LIN {X 0,Y 314.247,Z 438.29,A -85,B 0,C 180,E1 -15747.116,E2 -15747.116} C_VEL
LIN {X 0,Y 313.392,Z 444.97,A -85,B 0,C 180,E1 -15749.358,E2 -15749.358} C_VEL
LIN {X 0,Y 312.88,Z 449.381,A -85,B 0,C 180,E1 -15751.288,E2 -15751.288} C_VEL
LIN {X 0,Y 312.504,Z 451.733,A -85,B 0,C 180,E1 -15752.578,E2 -15752.578} C_VEL
LIN {X 0,Y 312.347,Z 453.646,A -85,B 0,C 180,E1 -15753.871,E2 -15753.871} C_VEL
LIN {X 0,Y 312.37,Z 455.131,A -85,B 0,C 180,E1 -15755.164,E2 -15755.164} C_VEL
LIN {X 0,Y 312.273,Z 456.882,A -85,B 0,C 180,E1 -15757.761,E2 -15757.761} C_VEL
LIN {X 0,Y 312.327,Z 457.191,A -85,B 0,C 180,E1 -15759.063,E2 -15759.063} C_VEL
LIN {X 0,Y 312.449,Z 457.109,A -85,B 0,C 180,E1 -15760.367,E2 -15760.367} C_VEL
LIN {X 0,Y 312.916,Z 455.702,A -85,B 0,C 180,E1 -15762.979,E2 -15762.979} C_VEL
LIN {X 0,Y 313.359,Z 454.404,A -85,B 0,C 180,E1 -15764.283,E2 -15764.283} C_VEL
LIN {X 0,Y 314.081,Z 451.635,A -85,B 0,C 180,E1 -15766.242,E2 -15766.242} C_VEL
LIN {X 0,Y 314.982,Z 447.824,A -85,B 0,C 180,E1 -15768.202,E2 -15768.202} C_VEL
LIN {X 0,Y 316.106,Z 442.855,A -85,B 0,C 180,E1 -15770.158,E2 -15770.158} C_VEL
LIN {X 0,Y 317.523,Z 436.525,A -85,B 0,C 180,E1 -15772.103,E2 -15772.103} C_VEL
LIN {X 0,Y 319.103,Z 428.554,A -85,B 0,C 180,E1 -15774.045,E2 -15774.045} C_VEL
LIN {X 0,Y 320.652,Z 420.359,A -85,B 0,C 180,E1 -15775.65,E2 -15775.65} C_VEL
LIN {X 0,Y 322.026,Z 411.372,A -85,B 0,C 180,E1 -15777.102,E2 -15777.102} C_VEL
LIN {X 0,Y 323.472,Z 401.574,A -85,B 0,C 180,E1 -15778.377,E2 -15778.377} C_VEL
LIN {X 0,Y 324.734,Z 390.84,A -85,B 0,C 180,E1 -15779.496,E2 -15779.496} C_VEL
LIN {X 0,Y 325.769,Z 379.701,A -85,B 0,C 180,E1 -15780.403,E2 -15780.403} C_VEL
LIN {X 0,Y 326.491,Z 366.602,A -85,B 0,C 180,E1 -15781.205,E2 -15781.205} C_VEL
LIN {X 0,Y 326.866,Z 354.631,A -85,B 0,C 180,E1 -15781.696,E2 -15781.696} C_VEL
LIN {X 0,Y 327.637,Z 314.685,A -85,B 0,C 180,E1 -15782.625,E2 -15782.625} C_VEL
LIN {X 0,Y 328.12,Z 297.79,A -85,B 0,C 180,E1 -15782.993,E2 -15782.993} C_VEL
LIN {X 0,Y 320.551,Z 282.248,A -85,B 0,C 180,E1 -15784.14,E2 -15784.14} C_VEL
LIN {X 0,Y 313.584,Z 269.449,A -85,B 0,C 180,E1 -15785.22,E2 -15785.22} C_VEL
LIN {X 0,Y 312.651,Z 267.172,A -85,B 0,C 180,E1 -15785.452,E2 -15785.452} C_VEL
LIN {X 0,Y 312.55,Z 266.564,A -85,B 0,C 180,E1 -15785.777,E2 -15785.777} C_VEL
LIN {X 0,Y 312.477,Z 266.546,A -85,B 0,C 180,E1 -15789.032,E2 -15789.032} C_VEL
LIN {X 0,Y 312.456,Z 266.549,A -85,B 0,C 180,E1 -15792.188,E2 -15792.188} C_VEL
LIN {X 0,Y 311.815,Z 266.64,A -85,B 0,C 180,E1 -15793.264,E2 -15793.264} C_VEL
LIN {X 0,Y 308.975,Z 266.996,A -85,B 0,C 180,E1 -15795.016,E2 -15795.016} C_VEL
LIN {X 0,Y 306.549,Z 267.286,A -85,B 0,C 180,E1 -15796.436,E2 -15796.436} C_VEL
LIN {X 0,Y 305.5,Z 267.412,A -85,B 0,C 180,E1 -15797.536,E2 -15797.536} C_VEL
LIN {X 0,Y 305.412,Z 267.426,A -85,B 0,C 180,E1 -15797.908,E2 -15797.908} C_VEL
LIN {X 0,Y 305.44,Z 267.414,A -85,B 0,C 180,E1 -15801.592,E2 -15801.592} C_VEL
LIN {X 0,Y 305.46,Z 267.432,A -85,B 0,C 180,E1 -15804.886,E2 -15804.886} C_VEL
LIN {X 0,Y 305.44,Z 267.41,A -85,B 0,C 180,E1 -15808.358,E2 -15808.358} C_VEL
LIN {X 0,Y 305.463,Z 267.41,A -85,B 0,C 180,E1 -15811.107,E2 -15811.107} C_VEL
LIN {X 0,Y 305.497,Z 267.433,A -85,B 0,C 180,E1 -15814.081,E2 -15814.081} C_VEL
LIN {X 0,Y 305.471,Z 267.395,A -85,B 0,C 180,E1 -15816.975,E2 -15816.975} C_VEL
LIN {X 0,Y 305.576,Z 267.413,A -85,B 0,C 180,E1 -15821.216,E2 -15821.216} C_VEL
LIN {X 0,Y 305.646,Z 267.399,A -85,B 0,C 180,E1 -15825.348,E2 -15825.348} C_VEL
LIN {X 0,Y 305.62,Z 267.409,A -85,B 0,C 180,E1 -15829.399,E2 -15829.399} C_VEL
LIN {X 0,Y 305.741,Z 267.394,A -85,B 0,C 180,E1 -15832.072,E2 -15832.072} C_VEL
LIN {X 0,Y 305.65,Z 267.407,A -85,B 0,C 180,E1 -15834.722,E2 -15834.722} C_VEL
LIN {X 0,Y 305.941,Z 267.374,A -85,B 0,C 180,E1 -15838.683,E2 -15838.683} C_VEL
LIN {X 0,Y 305.93,Z 267.364,A -85,B 0,C 180,E1 -15841.316,E2 -15841.316} C_VEL
LIN {X 0,Y 305.654,Z 267.412,A -85,B 0,C 180,E1 -15845.277,E2 -15845.277} C_VEL
LIN {X 0,Y 305.74,Z 267.387,A -85,B 0,C 180,E1 -15847.927,E2 -15847.927} C_VEL
LIN {X 0,Y 305.592,Z 267.41,A -85,B 0,C 180,E1 -15851.945,E2 -15851.945} C_VEL
LIN {X 0,Y 305.604,Z 267.414,A -85,B 0,C 180,E1 -15855.014,E2 -15855.014} C_VEL
LIN {X 0,Y 305.542,Z 267.425,A -85,B 0,C 180,E1 -15859.428,E2 -15859.428} C_VEL
LIN {X 0,Y 305.483,Z 267.429,A -85,B 0,C 180,E1 -15863.039,E2 -15863.039} C_VEL
LIN {X 0,Y 305.463,Z 267.419,A -85,B 0,C 180,E1 -15866.196,E2 -15866.196} C_VEL
LIN {X 0,Y 305.419,Z 267.425,A -85,B 0,C 180,E1 -15869.025,E2 -15869.025} C_VEL
LIN {X 0,Y 305.431,Z 267.435,A -85,B 0,C 180,E1 -15871.953,E2 -15871.953} C_VEL
LIN {X 0,Y 305.458,Z 267.424,A -85,B 0,C 180,E1 -15875.114,E2 -15875.114} C_VEL
LIN {X 0,Y 305.43,Z 267.426,A -85,B 0,C 180,E1 -15878.525,E2 -15878.525} C_VEL
LIN {X 0,Y 305.431,Z 267.431,A -85,B 0,C 180,E1 -15882.581,E2 -15882.581} C_VEL
LIN {X 0,Y 305.418,Z 267.433,A -85,B 0,C 180,E1 -15886.344,E2 -15886.344} C_VEL
LIN {X 0,Y 305.466,Z 267.601,A -85,B 0,C 180,E1 -15890.617,E2 -15890.617} C_VEL
LIN {X 0,Y 308.864,Z 279.639,A -85,B 0,C 180,E1 -15894.049,E2 -15894.049} C_VEL
LIN {X 0,Y 311.517,Z 290.832,A -85,B 0,C 180,E1 -15896.979,E2 -15896.979} C_VEL
LIN {X 0,Y 313.244,Z 300.295,A -85,B 0,C 180,E1 -15899.308,E2 -15899.308} C_VEL
LIN {X 0,Y 311.503,Z 313.167,A -85,B 0,C 180,E1 -15902.016,E2 -15902.016} C_VEL
LIN {X 0,Y 311.73,Z 315.517,A -85,B 0,C 180,E1 -15902.182,E2 -15902.182} C_VEL
LIN {X 0,Y 316.099,Z 342.071,A -85,B 0,C 180,E1 -15903.321,E2 -15903.321} C_VEL
LIN {X 0,Y 319.329,Z 367.742,A -85,B 0,C 180,E1 -15904.287,E2 -15904.287} C_VEL
LIN {X 0,Y 319.905,Z 376.948,A -85,B 0,C 180,E1 -15904.572,E2 -15904.572} C_VEL
LIN {X 0,Y 318.499,Z 425.443,A -85,B 0,C 180,E1 -15905.69,E2 -15905.69} C_VEL
LIN {X 0,Y 317.484,Z 439.253,A -85,B 0,C 180,E1 -15906.259,E2 -15906.259} C_VEL
LIN {X 0,Y 316.086,Z 451.686,A -85,B 0,C 180,E1 -15907.015,E2 -15907.015} C_VEL
LIN {X 0,Y 314.257,Z 463.613,A -85,B 0,C 180,E1 -15908.001,E2 -15908.001} C_VEL
LIN {X 0,Y 312.257,Z 475.089,A -85,B 0,C 180,E1 -15909.238,E2 -15909.238} C_VEL
LIN {X 0,Y 310.326,Z 485.479,A -85,B 0,C 180,E1 -15910.657,E2 -15910.657} C_VEL
LIN {X 0,Y 308.647,Z 494.011,A -85,B 0,C 180,E1 -15912.097,E2 -15912.097} C_VEL
LIN {X 0,Y 306.953,Z 503.327,A -85,B 0,C 180,E1 -15914.053,E2 -15914.053} C_VEL
LIN {X 0,Y 305.899,Z 509.739,A -85,B 0,C 180,E1 -15915.701,E2 -15915.701} C_VEL
LIN {X 0,Y 304.737,Z 516.994,A -85,B 0,C 180,E1 -15918.02,E2 -15918.02} C_VEL
LIN {X 0,Y 304.214,Z 521.881,A -85,B 0,C 180,E1 -15920.022,E2 -15920.022} C_VEL
LIN {X 0,Y 304.081,Z 525.679,A -85,B 0,C 180,E1 -15922.029,E2 -15922.029} C_VEL
LIN {X 0,Y 304.187,Z 527.793,A -85,B 0,C 180,E1 -15923.454,E2 -15923.454} C_VEL
LIN {X 0,Y 304.482,Z 530.322,A -85,B 0,C 180,E1 -15926.029,E2 -15926.029} C_VEL
LIN {X 0,Y 304.663,Z 531.039,A -85,B 0,C 180,E1 -15927.355,E2 -15927.355} C_VEL
LIN {X 0,Y 304.672,Z 531.334,A -85,B 0,C 180,E1 -15928.678,E2 -15928.678} C_VEL
LIN {X 0,Y 304.795,Z 531.2,A -85,B 0,C 180,E1 -15929.999,E2 -15929.999} C_VEL
LIN {X 0,Y 304.732,Z 530.624,A -85,B 0,C 180,E1 -15931.321,E2 -15931.321} C_VEL
LIN {X 0,Y 304.731,Z 529.649,A -85,B 0,C 180,E1 -15932.643,E2 -15932.643} C_VEL
LIN {X 0,Y 304.622,Z 528.244,A -85,B 0,C 180,E1 -15933.968,E2 -15933.968} C_VEL
LIN {X 0,Y 304.391,Z 525.237,A -85,B 0,C 180,E1 -15935.963,E2 -15935.963} C_VEL
LIN {X 0,Y 304.244,Z 521.148,A -85,B 0,C 180,E1 -15937.966,E2 -15937.966} C_VEL
LIN {X 0,Y 304.376,Z 514.864,A -85,B 0,C 180,E1 -15940.308,E2 -15940.308} C_VEL
LIN {X 0,Y 304.867,Z 508.012,A -85,B 0,C 180,E1 -15942.311,E2 -15942.311} C_VEL
LIN {X 0,Y 305.704,Z 499.529,A -85,B 0,C 180,E1 -15944.307,E2 -15944.307} C_VEL
LIN {X 0,Y 306.686,Z 490.83,A -85,B 0,C 180,E1 -15945.961,E2 -15945.961} C_VEL
LIN {X 0,Y 307.809,Z 481.296,A -85,B 0,C 180,E1 -15947.437,E2 -15947.437} C_VEL
LIN {X 0,Y 309.296,Z 469.516,A -85,B 0,C 180,E1 -15948.892,E2 -15948.892} C_VEL
LIN {X 0,Y 310.641,Z 457.868,A -85,B 0,C 180,E1 -15950.009,E2 -15950.009} C_VEL
LIN {X 0,Y 311.816,Z 445.781,A -85,B 0,C 180,E1 -15950.878,E2 -15950.878} C_VEL
LIN {X 0,Y 312.673,Z 432.658,A -85,B 0,C 180,E1 -15951.552,E2 -15951.552} C_VEL
LIN {X 0,Y 313.184,Z 420.288,A -85,B 0,C 180,E1 -15951.947,E2 -15951.947} C_VEL
LIN {X 0,Y 313.933,Z 371.708,A -85,B 0,C 180,E1 -15953.054,E2 -15953.054} C_VEL
LIN {X 0,Y 309.351,Z 325.296,A -85,B 0,C 180,E1 -15954.472,E2 -15954.472} C_VEL
LIN {X 0,Y 308.185,Z 315.1,A -85,B 0,C 180,E1 -15954.851,E2 -15954.851} C_VEL
LIN {X 0,Y 310.188,Z 295.934,A -85,B 0,C 180,E1 -15958.78,E2 -15958.78} C_VEL
LIN {X 0,Y 310.465,Z 290.771,A -85,B 0,C 180,E1 -15959.867,E2 -15959.867} C_VEL
LIN {X 0,Y 307.511,Z 276.202,A -85,B 0,C 180,E1 -15963.263,E2 -15963.263} C_VEL
LIN {X 0,Y 305.499,Z 267.537,A -85,B 0,C 180,E1 -15965.435,E2 -15965.435} C_VEL
LIN {X 0,Y 305.428,Z 267.433,A -85,B 0,C 180,E1 -15968.524,E2 -15968.524} C_VEL
LIN {X 0,Y 305.428,Z 267.439,A -85,B 0,C 180,E1 -15972.58,E2 -15972.58} C_VEL
LIN {X 0,Y 305.413,Z 267.431,A -85,B 0,C 180,E1 -15976.343,E2 -15976.343} C_VEL
LIN {X 0,Y 305.402,Z 267.44,A -85,B 0,C 180,E1 -15979.884,E2 -15979.884} C_VEL
LIN {X 0,Y 305.454,Z 267.435,A -85,B 0,C 180,E1 -15983.636,E2 -15983.636} C_VEL
LIN {X 0,Y 305.455,Z 267.433,A -85,B 0,C 180,E1 -15986.482,E2 -15986.482} C_VEL
LIN {X 0,Y 305.407,Z 267.44,A -85,B 0,C 180,E1 -15989.585,E2 -15989.585} C_VEL
LIN {X 0,Y 305.444,Z 267.437,A -85,B 0,C 180,E1 -15992.601,E2 -15992.601} C_VEL
LIN {X 0,Y 305.463,Z 267.43,A -85,B 0,C 180,E1 -15995.535,E2 -15995.535} C_VEL
LIN {X 0,Y 305.451,Z 267.436,A -85,B 0,C 180,E1 -15998.399,E2 -15998.399} C_VEL
LIN {X 0,Y 305.525,Z 267.421,A -85,B 0,C 180,E1 -16002.6,E2 -16002.6} C_VEL
LIN {X 0,Y 305.616,Z 267.414,A -85,B 0,C 180,E1 -16005.348,E2 -16005.348} C_VEL
LIN {X 0,Y 305.613,Z 267.408,A -85,B 0,C 180,E1 -16009.399,E2 -16009.399} C_VEL
LIN {X 0,Y 305.734,Z 267.395,A -85,B 0,C 180,E1 -16012.073,E2 -16012.073} C_VEL
LIN {X 0,Y 305.647,Z 267.414,A -85,B 0,C 180,E1 -16014.723,E2 -16014.723} C_VEL
LIN {X 0,Y 305.924,Z 267.37,A -85,B 0,C 180,E1 -16018.684,E2 -16018.684} C_VEL
LIN {X 0,Y 305.933,Z 267.371,A -85,B 0,C 180,E1 -16021.317,E2 -16021.317} C_VEL
LIN {X 0,Y 305.773,Z 267.392,A -85,B 0,C 180,E1 -16026.599,E2 -16026.599} C_VEL
LIN {X 0,Y 305.674,Z 267.399,A -85,B 0,C 180,E1 -16029.262,E2 -16029.262} C_VEL
LIN {X 0,Y 305.575,Z 267.418,A -85,B 0,C 180,E1 -16033.297,E2 -16033.297} C_VEL
LIN {X 0,Y 305.541,Z 267.423,A -85,B 0,C 180,E1 -16036.023,E2 -16036.023} C_VEL
LIN {X 0,Y 305.475,Z 267.433,A -85,B 0,C 180,E1 -16040.188,E2 -16040.188} C_VEL
LIN {X 0,Y 305.447,Z 267.432,A -85,B 0,C 180,E1 -16044.467,E2 -16044.467} C_VEL
LIN {X 0,Y 305.432,Z 267.433,A -85,B 0,C 180,E1 -16047.401,E2 -16047.401} C_VEL
LIN {X 0,Y 305.409,Z 267.441,A -85,B 0,C 180,E1 -16050.415,E2 -16050.415} C_VEL
LIN {X 0,Y 305.458,Z 267.432,A -85,B 0,C 180,E1 -16054.079,E2 -16054.079} C_VEL
LIN {X 0,Y 305.445,Z 267.435,A -85,B 0,C 180,E1 -16056.744,E2 -16056.744} C_VEL
LIN {X 0,Y 305.403,Z 267.432,A -85,B 0,C 180,E1 -16060.591,E2 -16060.591} C_VEL
LIN {X 0,Y 305.415,Z 267.421,A -85,B 0,C 180,E1 -16063.658,E2 -16063.658} C_VEL
LIN {X 0,Y 305.43,Z 267.438,A -85,B 0,C 180,E1 -16067.42,E2 -16067.42} C_VEL
LIN {X 0,Y 305.438,Z 267.428,A -85,B 0,C 180,E1 -16071.594,E2 -16071.594} C_VEL
LIN {X 0,Y 305.459,Z 267.43,A -85,B 0,C 180,E1 -16074.888,E2 -16074.888} C_VEL
LIN {X 0,Y 305.437,Z 267.433,A -85,B 0,C 180,E1 -16078.361,E2 -16078.361} C_VEL
LIN {X 0,Y 305.449,Z 267.431,A -85,B 0,C 180,E1 -16081.108,E2 -16081.108} C_VEL
LIN {X 0,Y 305.478,Z 267.428,A -85,B 0,C 180,E1 -16084.081,E2 -16084.081} C_VEL
LIN {X 0,Y 305.456,Z 267.433,A -85,B 0,C 180,E1 -16088.401,E2 -16088.401} C_VEL
LIN {X 0,Y 305.5,Z 267.401,A -85,B 0,C 180,E1 -16091.213,E2 -16091.213} C_VEL
LIN {X 0,Y 305.528,Z 267.629,A -85,B 0,C 180,E1 -16093.45,E2 -16093.45} C_VEL
LIN {X 0,Y 305.832,Z 268.784,A -85,B 0,C 180,E1 -16093.661,E2 -16093.661} C_VEL
LIN {X 0,Y 314.272,Z 288.888,A -85,B 0,C 180,E1 -16094.778,E2 -16094.778} C_VEL
LIN {X 0,Y 315.387,Z 291.963,A -85,B 0,C 180,E1 -16094.93,E2 -16094.93} C_VEL
LIN {X 0,Y 314.323,Z 354.388,A -85,B 0,C 180,E1 -16096.373,E2 -16096.373} C_VEL
LIN {X 0,Y 313.978,Z 367.298,A -85,B 0,C 180,E1 -16096.917,E2 -16096.917} C_VEL
LIN {X 0,Y 313.505,Z 379.756,A -85,B 0,C 180,E1 -16097.705,E2 -16097.705} C_VEL
LIN {X 0,Y 312.674,Z 391.136,A -85,B 0,C 180,E1 -16098.658,E2 -16098.658} C_VEL
LIN {X 0,Y 311.574,Z 402.813,A -85,B 0,C 180,E1 -16099.933,E2 -16099.933} C_VEL
LIN {X 0,Y 310.555,Z 413.216,A -85,B 0,C 180,E1 -16101.378,E2 -16101.378} C_VEL
LIN {X 0,Y 309.377,Z 423.453,A -85,B 0,C 180,E1 -16103.151,E2 -16103.151} C_VEL
LIN {X 0,Y 308.236,Z 432.34,A -85,B 0,C 180,E1 -16105.096,E2 -16105.096} C_VEL
LIN {X 0,Y 307.228,Z 439.521,A -85,B 0,C 180,E1 -16107.05,E2 -16107.05} C_VEL
LIN {X 0,Y 306.348,Z 446.095,A -85,B 0,C 180,E1 -16109.343,E2 -16109.343} C_VEL
LIN {X 0,Y 305.811,Z 450.446,A -85,B 0,C 180,E1 -16111.317,E2 -16111.317} C_VEL
LIN {X 0,Y 305.442,Z 452.767,A -85,B 0,C 180,E1 -16112.638,E2 -16112.638} C_VEL
LIN {X 0,Y 305.298,Z 454.65,A -85,B 0,C 180,E1 -16113.96,E2 -16113.96} C_VEL
LIN {X 0,Y 305.317,Z 456.082,A -85,B 0,C 180,E1 -16115.283,E2 -16115.283} C_VEL
LIN {X 0,Y 305.243,Z 457.776,A -85,B 0,C 180,E1 -16117.941,E2 -16117.941} C_VEL
LIN {X 0,Y 305.304,Z 458.059,A -85,B 0,C 180,E1 -16119.273,E2 -16119.273} C_VEL
LIN {X 0,Y 305.457,Z 457.922,A -85,B 0,C 180,E1 -16120.607,E2 -16120.607} C_VEL
LIN {X 0,Y 305.96,Z 456.46,A -85,B 0,C 180,E1 -16123.28,E2 -16123.28} C_VEL
LIN {X 0,Y 306.433,Z 455.132,A -85,B 0,C 180,E1 -16124.613,E2 -16124.613} C_VEL
LIN {X 0,Y 307.192,Z 452.307,A -85,B 0,C 180,E1 -16126.617,E2 -16126.617} C_VEL
LIN {X 0,Y 308.169,Z 448.433,A -85,B 0,C 180,E1 -16128.619,E2 -16128.619} C_VEL
LIN {X 0,Y 309.397,Z 443.38,A -85,B 0,C 180,E1 -16130.615,E2 -16130.615} C_VEL
LIN {X 0,Y 310.889,Z 436.95,A -85,B 0,C 180,E1 -16132.601,E2 -16132.601} C_VEL
LIN {X 0,Y 312.574,Z 428.89,A -85,B 0,C 180,E1 -16134.58,E2 -16134.58} C_VEL
LIN {X 0,Y 314.186,Z 420.657,A -85,B 0,C 180,E1 -16136.205,E2 -16136.205} C_VEL
LIN {X 0,Y 315.683,Z 411.474,A -85,B 0,C 180,E1 -16137.693,E2 -16137.693} C_VEL
LIN {X 0,Y 317.115,Z 401.452,A -85,B 0,C 180,E1 -16138.999,E2 -16138.999} C_VEL
LIN {X 0,Y 318.507,Z 390.466,A -85,B 0,C 180,E1 -16140.132,E2 -16140.132} C_VEL
LIN {X 0,Y 319.526,Z 379.515,A -85,B 0,C 180,E1 -16141.019,E2 -16141.019} C_VEL
LIN {X 0,Y 320.249,Z 366.514,A -85,B 0,C 180,E1 -16141.811,E2 -16141.811} C_VEL
LIN {X 0,Y 320.628,Z 354.436,A -85,B 0,C 180,E1 -16142.291,E2 -16142.291} C_VEL
LIN {X 0,Y 321.455,Z 314.337,A -85,B 0,C 180,E1 -16143.234,E2 -16143.234} C_VEL
LIN {X 0,Y 321.851,Z 299.831,A -85,B 0,C 180,E1 -16143.56,E2 -16143.56} C_VEL
LIN {X 0,Y 313.661,Z 283.186,A -85,B 0,C 180,E1 -16144.849,E2 -16144.849} C_VEL
LIN {X 0,Y 306.731,Z 270.599,A -85,B 0,C 180,E1 -16145.968,E2 -16145.968} C_VEL
LIN {X 0,Y 305.602,Z 268.05,A -85,B 0,C 180,E1 -16146.239,E2 -16146.239} C_VEL
LIN {X 0,Y 305.49,Z 267.483,A -85,B 0,C 180,E1 -16146.493,E2 -16146.493} C_VEL
LIN {X 0,Y 305.41,Z 267.446,A -85,B 0,C 180,E1 -16150.115,E2 -16150.115} C_VEL
LIN {X 0,Y 305.42,Z 267.44,A -85,B 0,C 180,E1 -16153.656,E2 -16153.656} C_VEL
LIN {X 0,Y 305.433,Z 267.419,A -85,B 0,C 180,E1 -16157.418,E2 -16157.418} C_VEL
LIN {X 0,Y 305.412,Z 267.426,A -85,B 0,C 180,E1 -16157.908,E2 -16157.908} C_VEL
LIN {X 0,Y 304.742,Z 267.525,A -85,B 0,C 180,E1 -16159.009,E2 -16159.009} C_VEL
LIN {X 0,Y 301.912,Z 267.865,A -85,B 0,C 180,E1 -16160.801,E2 -16160.801} C_VEL
LIN {X 0,Y 299.516,Z 268.151,A -85,B 0,C 180,E1 -16162.255,E2 -16162.255} C_VEL
LIN {X 0,Y 298.488,Z 268.279,A -85,B 0,C 180,E1 -16163.38,E2 -16163.38} C_VEL
LIN {X 0,Y 298.403,Z 268.294,A -85,B 0,C 180,E1 -16163.761,E2 -16163.761} C_VEL
LIN {X 0,Y 298.391,Z 268.308,A -85,B 0,C 180,E1 -16167.199,E2 -16167.199} C_VEL
LIN {X 0,Y 298.369,Z 268.286,A -85,B 0,C 180,E1 -16170.635,E2 -16170.635} C_VEL
LIN {X 0,Y 298.436,Z 268.307,A -85,B 0,C 180,E1 -16174.919,E2 -16174.919} C_VEL
LIN {X 0,Y 298.401,Z 268.266,A -85,B 0,C 180,E1 -16177.862,E2 -16177.862} C_VEL
LIN {X 0,Y 298.522,Z 268.281,A -85,B 0,C 180,E1 -16180.755,E2 -16180.755} C_VEL
LIN {X 0,Y 298.59,Z 268.279,A -85,B 0,C 180,E1 -16184.994,E2 -16184.994} C_VEL
LIN {X 0,Y 298.579,Z 268.29,A -85,B 0,C 180,E1 -16189.146,E2 -16189.146} C_VEL
LIN {X 0,Y 298.693,Z 268.269,A -85,B 0,C 180,E1 -16191.884,E2 -16191.884} C_VEL
LIN {X 0,Y 298.62,Z 268.283,A -85,B 0,C 180,E1 -16194.598,E2 -16194.598} C_VEL
LIN {X 0,Y 298.907,Z 268.251,A -85,B 0,C 180,E1 -16198.652,E2 -16198.652} C_VEL
LIN {X 0,Y 298.898,Z 268.239,A -85,B 0,C 180,E1 -16201.347,E2 -16201.347} C_VEL
LIN {X 0,Y 298.727,Z 268.263,A -85,B 0,C 180,E1 -16206.755,E2 -16206.755} C_VEL
LIN {X 0,Y 298.621,Z 268.284,A -85,B 0,C 180,E1 -16209.482,E2 -16209.482} C_VEL
LIN {X 0,Y 298.539,Z 268.285,A -85,B 0,C 180,E1 -16213.616,E2 -16213.616} C_VEL
LIN {X 0,Y 298.483,Z 268.303,A -85,B 0,C 180,E1 -16216.412,E2 -16216.412} C_VEL
LIN {X 0,Y 298.482,Z 268.307,A -85,B 0,C 180,E1 -16219.641,E2 -16219.641} C_VEL
LIN {X 0,Y 298.416,Z 268.316,A -85,B 0,C 180,E1 -16223.601,E2 -16223.601} C_VEL
LIN {X 0,Y 298.402,Z 268.292,A -85,B 0,C 180,E1 -16226.583,E2 -16226.583} C_VEL
LIN {X 0,Y 298.352,Z 268.314,A -85,B 0,C 180,E1 -16229.648,E2 -16229.648} C_VEL
LIN {X 0,Y 298.388,Z 268.3,A -85,B 0,C 180,E1 -16232.801,E2 -16232.801} C_VEL
LIN {X 0,Y 298.401,Z 268.315,A -85,B 0,C 180,E1 -16236.072,E2 -16236.072} C_VEL
LIN {X 0,Y 298.371,Z 268.306,A -85,B 0,C 180,E1 -16239.492,E2 -16239.492} C_VEL
LIN {X 0,Y 298.366,Z 268.308,A -85,B 0,C 180,E1 -16243.097,E2 -16243.097} C_VEL
LIN {X 0,Y 298.367,Z 268.311,A -85,B 0,C 180,E1 -16246.915,E2 -16246.915} C_VEL
LIN {X 0,Y 298.413,Z 268.534,A -85,B 0,C 180,E1 -16249.912,E2 -16249.912} C_VEL
LIN {X 0,Y 301.837,Z 280.529,A -85,B 0,C 180,E1 -16253.445,E2 -16253.445} C_VEL
LIN {X 0,Y 304.446,Z 291.278,A -85,B 0,C 180,E1 -16256.356,E2 -16256.356} C_VEL
LIN {X 0,Y 306.43,Z 301.402,A -85,B 0,C 180,E1 -16258.933,E2 -16258.933} C_VEL
LIN {X 0,Y 305.149,Z 311.226,A -85,B 0,C 180,E1 -16261.075,E2 -16261.075} C_VEL
LIN {X 0,Y 305.001,Z 313.048,A -85,B 0,C 180,E1 -16261.364,E2 -16261.364} C_VEL
LIN {X 0,Y 309.751,Z 342.135,A -85,B 0,C 180,E1 -16262.671,E2 -16262.671} C_VEL
LIN {X 0,Y 312.825,Z 366.354,A -85,B 0,C 180,E1 -16263.617,E2 -16263.617} C_VEL
LIN {X 0,Y 313.654,Z 376.711,A -85,B 0,C 180,E1 -16263.965,E2 -16263.965} C_VEL
LIN {X 0,Y 312.216,Z 424.344,A -85,B 0,C 180,E1 -16265.08,E2 -16265.08} C_VEL
LIN {X 0,Y 311.17,Z 438.229,A -85,B 0,C 180,E1 -16265.658,E2 -16265.658} C_VEL
LIN {X 0,Y 309.71,Z 450.709,A -85,B 0,C 180,E1 -16266.425,E2 -16266.425} C_VEL
LIN {X 0,Y 307.92,Z 461.867,A -85,B 0,C 180,E1 -16267.346,E2 -16267.346} C_VEL
LIN {X 0,Y 305.849,Z 473.5,A -85,B 0,C 180,E1 -16268.605,E2 -16268.605} C_VEL
LIN {X 0,Y 303.846,Z 484.01,A -85,B 0,C 180,E1 -16270.052,E2 -16270.052} C_VEL
LIN {X 0,Y 301.881,Z 493.523,A -85,B 0,C 180,E1 -16271.682,E2 -16271.682} C_VEL
LIN {X 0,Y 300.097,Z 502.756,A -85,B 0,C 180,E1 -16273.678,E2 -16273.678} C_VEL
LIN {X 0,Y 298.736,Z 510.255,A -85,B 0,C 180,E1 -16275.698,E2 -16275.698} C_VEL
LIN {X 0,Y 297.757,Z 516.325,A -85,B 0,C 180,E1 -16277.735,E2 -16277.735} C_VEL
LIN {X 0,Y 297.159,Z 521.169,A -85,B 0,C 180,E1 -16279.783,E2 -16279.783} C_VEL
LIN {X 0,Y 297.013,Z 524.932,A -85,B 0,C 180,E1 -16281.838,E2 -16281.838} C_VEL
LIN {X 0,Y 297.124,Z 527.171,A -85,B 0,C 180,E1 -16283.435,E2 -16283.435} C_VEL
LIN {X 0,Y 297.397,Z 529.508,A -85,B 0,C 180,E1 -16285.934,E2 -16285.934} C_VEL
LIN {X 0,Y 297.613,Z 530.213,A -85,B 0,C 180,E1 -16287.292,E2 -16287.292} C_VEL
LIN {X 0,Y 297.622,Z 530.486,A -85,B 0,C 180,E1 -16288.646,E2 -16288.646} C_VEL
LIN {X 0,Y 297.747,Z 530.325,A -85,B 0,C 180,E1 -16289.999,E2 -16289.999} C_VEL
LIN {X 0,Y 297.682,Z 529.732,A -85,B 0,C 180,E1 -16291.352,E2 -16291.352} C_VEL
LIN {X 0,Y 297.682,Z 528.739,A -85,B 0,C 180,E1 -16292.706,E2 -16292.706} C_VEL
LIN {X 0,Y 297.553,Z 527.306,A -85,B 0,C 180,E1 -16294.063,E2 -16294.063} C_VEL
LIN {X 0,Y 297.281,Z 523.757,A -85,B 0,C 180,E1 -16296.382,E2 -16296.382} C_VEL
LIN {X 0,Y 297.162,Z 518.474,A -85,B 0,C 180,E1 -16298.842,E2 -16298.842} C_VEL
LIN {X 0,Y 297.4,Z 512.745,A -85,B 0,C 180,E1 -16300.897,E2 -16300.897} C_VEL
LIN {X 0,Y 297.951,Z 505.605,A -85,B 0,C 180,E1 -16302.948,E2 -16302.948} C_VEL
LIN {X 0,Y 298.705,Z 498.328,A -85,B 0,C 180,E1 -16304.65,E2 -16304.65} C_VEL
LIN {X 0,Y 299.834,Z 489.552,A -85,B 0,C 180,E1 -16306.335,E2 -16306.335} C_VEL
LIN {X 0,Y 301.053,Z 479.94,A -85,B 0,C 180,E1 -16307.841,E2 -16307.841} C_VEL
LIN {X 0,Y 302.362,Z 469.485,A -85,B 0,C 180,E1 -16309.166,E2 -16309.166} C_VEL
LIN {X 0,Y 303.728,Z 458.06,A -85,B 0,C 180,E1 -16310.308,E2 -16310.308} C_VEL
LIN {X 0,Y 304.948,Z 446.418,A -85,B 0,C 180,E1 -16311.194,E2 -16311.194} C_VEL
LIN {X 0,Y 305.869,Z 432.974,A -85,B 0,C 180,E1 -16311.923,E2 -16311.923} C_VEL
LIN {X 0,Y 306.457,Z 419.843,A -85,B 0,C 180,E1 -16312.366,E2 -16312.366} C_VEL
LIN {X 0,Y 307.263,Z 372.556,A -85,B 0,C 180,E1 -16313.465,E2 -16313.465} C_VEL
LIN {X 0,Y 302.775,Z 326.508,A -85,B 0,C 180,E1 -16314.91,E2 -16314.91} C_VEL
LIN {X 0,Y 301.342,Z 314.336,A -85,B 0,C 180,E1 -16315.35,E2 -16315.35} C_VEL
LIN {X 0,Y 303.309,Z 296.361,A -85,B 0,C 180,E1 -16319.115,E2 -16319.115} C_VEL
LIN {X 0,Y 303.6,Z 292.938,A -85,B 0,C 180,E1 -16319.847,E2 -16319.847} C_VEL
LIN {X 0,Y 301.035,Z 279.672,A -85,B 0,C 180,E1 -16322.991,E2 -16322.991} C_VEL
LIN {X 0,Y 298.495,Z 268.452,A -85,B 0,C 180,E1 -16325.832,E2 -16325.832} C_VEL
LIN {X 0,Y 298.368,Z 268.308,A -85,B 0,C 180,E1 -16329.491,E2 -16329.491} C_VEL
LIN {X 0,Y 298.363,Z 268.316,A -85,B 0,C 180,E1 -16333.096,E2 -16333.096} C_VEL
LIN {X 0,Y 298.362,Z 268.312,A -85,B 0,C 180,E1 -16336.914,E2 -16336.914} C_VEL
LIN {X 0,Y 298.377,Z 268.315,A -85,B 0,C 180,E1 -16341.01,E2 -16341.01} C_VEL
LIN {X 0,Y 298.396,Z 268.314,A -85,B 0,C 180,E1 -16343.927,E2 -16343.927} C_VEL
LIN {X 0,Y 298.383,Z 268.309,A -85,B 0,C 180,E1 -16347.198,E2 -16347.198} C_VEL
LIN {X 0,Y 298.396,Z 268.313,A -85,B 0,C 180,E1 -16351.898,E2 -16351.898} C_VEL
LIN {X 0,Y 298.428,Z 268.306,A -85,B 0,C 180,E1 -16354.919,E2 -16354.919} C_VEL
LIN {X 0,Y 298.389,Z 268.314,A -85,B 0,C 180,E1 -16357.861,E2 -16357.861} C_VEL
LIN {X 0,Y 298.453,Z 268.304,A -85,B 0,C 180,E1 -16360.751,E2 -16360.751} C_VEL
LIN {X 0,Y 298.577,Z 268.294,A -85,B 0,C 180,E1 -16364.994,E2 -16364.994} C_VEL
LIN {X 0,Y 298.572,Z 268.285,A -85,B 0,C 180,E1 -16369.146,E2 -16369.146} C_VEL
LIN {X 0,Y 298.686,Z 268.272,A -85,B 0,C 180,E1 -16371.884,E2 -16371.884} C_VEL
LIN {X 0,Y 298.616,Z 268.29,A -85,B 0,C 180,E1 -16374.598,E2 -16374.598} C_VEL
LIN {X 0,Y 298.892,Z 268.245,A -85,B 0,C 180,E1 -16378.653,E2 -16378.653} C_VEL
LIN {X 0,Y 298.9,Z 268.247,A -85,B 0,C 180,E1 -16381.348,E2 -16381.348} C_VEL
LIN {X 0,Y 298.721,Z 268.269,A -85,B 0,C 180,E1 -16386.756,E2 -16386.756} C_VEL
LIN {X 0,Y 298.607,Z 268.279,A -85,B 0,C 180,E1 -16389.483,E2 -16389.483} C_VEL
LIN {X 0,Y 298.534,Z 268.296,A -85,B 0,C 180,E1 -16393.617,E2 -16393.617} C_VEL
LIN {X 0,Y 298.474,Z 268.297,A -85,B 0,C 180,E1 -16396.413,E2 -16396.413} C_VEL
LIN {X 0,Y 298.433,Z 268.305,A -85,B 0,C 180,E1 -16399.617,E2 -16399.617} C_VEL
LIN {X 0,Y 298.38,Z 268.315,A -85,B 0,C 180,E1 -16403.605,E2 -16403.605} C_VEL
LIN {X 0,Y 298.393,Z 268.31,A -85,B 0,C 180,E1 -16406.584,E2 -16406.584} C_VEL
LIN {X 0,Y 298.349,Z 268.321,A -85,B 0,C 180,E1 -16409.649,E2 -16409.649} C_VEL
LIN {X 0,Y 298.386,Z 268.309,A -85,B 0,C 180,E1 -16412.802,E2 -16412.802} C_VEL
LIN {X 0,Y 298.397,Z 268.317,A -85,B 0,C 180,E1 -16416.073,E2 -16416.073} C_VEL
LIN {X 0,Y 298.368,Z 268.317,A -85,B 0,C 180,E1 -16419.493,E2 -16419.493} C_VEL
LIN {X 0,Y 298.364,Z 268.295,A -85,B 0,C 180,E1 -16423.098,E2 -16423.098} C_VEL
LIN {X 0,Y 298.365,Z 268.315,A -85,B 0,C 180,E1 -16426.916,E2 -16426.916} C_VEL
LIN {X 0,Y 298.382,Z 268.311,A -85,B 0,C 180,E1 -16431.012,E2 -16431.012} C_VEL
LIN {X 0,Y 298.401,Z 268.304,A -85,B 0,C 180,E1 -16433.929,E2 -16433.929} C_VEL
LIN {X 0,Y 298.39,Z 268.317,A -85,B 0,C 180,E1 -16437.201,E2 -16437.201} C_VEL
LIN {X 0,Y 298.361,Z 268.311,A -85,B 0,C 180,E1 -16440.64,E2 -16440.64} C_VEL
LIN {X 0,Y 298.421,Z 268.305,A -85,B 0,C 180,E1 -16444.919,E2 -16444.919} C_VEL
LIN {X 0,Y 298.39,Z 268.314,A -85,B 0,C 180,E1 -16447.862,E2 -16447.862} C_VEL
LIN {X 0,Y 298.451,Z 268.276,A -85,B 0,C 180,E1 -16450.752,E2 -16450.752} C_VEL
LIN {X 0,Y 298.488,Z 268.573,A -85,B 0,C 180,E1 -16452.947,E2 -16452.947} C_VEL
LIN {X 0,Y 298.719,Z 269.516,A -85,B 0,C 180,E1 -16453.123,E2 -16453.123} C_VEL
LIN {X 0,Y 306.932,Z 288.664,A -85,B 0,C 180,E1 -16454.244,E2 -16454.244} C_VEL
LIN {X 0,Y 308.831,Z 294.105,A -85,B 0,C 180,E1 -16454.516,E2 -16454.516} C_VEL
LIN {X 0,Y 307.644,Z 354.477,A -85,B 0,C 180,E1 -16455.932,E2 -16455.932} C_VEL
LIN {X 0,Y 307.311,Z 367.077,A -85,B 0,C 180,E1 -16456.452,E2 -16456.452} C_VEL
LIN {X 0,Y 306.837,Z 379.906,A -85,B 0,C 180,E1 -16457.265,E2 -16457.265} C_VEL
LIN {X 0,Y 305.958,Z 391.442,A -85,B 0,C 180,E1 -16458.238,E2 -16458.238} C_VEL
LIN {X 0,Y 304.963,Z 401.962,A -85,B 0,C 180,E1 -16459.377,E2 -16459.377} C_VEL
LIN {X 0,Y 303.832,Z 412.695,A -85,B 0,C 180,E1 -16460.85,E2 -16460.85} C_VEL
LIN {X 0,Y 302.862,Z 421.434,A -85,B 0,C 180,E1 -16462.333,E2 -16462.333} C_VEL
LIN {X 0,Y 301.603,Z 430.949,A -85,B 0,C 180,E1 -16464.317,E2 -16464.317} C_VEL
LIN {X 0,Y 300.468,Z 438.559,A -85,B 0,C 180,E1 -16466.313,E2 -16466.313} C_VEL
LIN {X 0,Y 299.519,Z 445.543,A -85,B 0,C 180,E1 -16468.656,E2 -16468.656} C_VEL
LIN {X 0,Y 298.943,Z 450.201,A -85,B 0,C 180,E1 -16470.674,E2 -16470.674} C_VEL
LIN {X 0,Y 298.381,Z 453.801,A -85,B 0,C 180,E1 -16472.701,E2 -16472.701} C_VEL
LIN {X 0,Y 298.248,Z 455.648,A -85,B 0,C 180,E1 -16474.054,E2 -16474.054} C_VEL
LIN {X 0,Y 298.252,Z 457.031,A -85,B 0,C 180,E1 -16475.409,E2 -16475.409} C_VEL
LIN {X 0,Y 298.199,Z 458.683,A -85,B 0,C 180,E1 -16478.161,E2 -16478.161} C_VEL
LIN {X 0,Y 298.287,Z 458.918,A -85,B 0,C 180,E1 -16479.493,E2 -16479.493} C_VEL
LIN {X 0,Y 298.68,Z 458.17,A -85,B 0,C 180,E1 -16482.227,E2 -16482.227} C_VEL
LIN {X 0,Y 299.012,Z 457.219,A -85,B 0,C 180,E1 -16483.594,E2 -16483.594} C_VEL
LIN {X 0,Y 299.976,Z 454.294,A -85,B 0,C 180,E1 -16486.141,E2 -16486.141} C_VEL
LIN {X 0,Y 301.017,Z 450.442,A -85,B 0,C 180,E1 -16488.373,E2 -16488.373} C_VEL
LIN {X 0,Y 302.207,Z 445.729,A -85,B 0,C 180,E1 -16490.416,E2 -16490.416} C_VEL
LIN {X 0,Y 303.685,Z 439.84,A -85,B 0,C 180,E1 -16492.408,E2 -16492.408} C_VEL
LIN {X 0,Y 305.412,Z 432.185,A -85,B 0,C 180,E1 -16494.469,E2 -16494.469} C_VEL
LIN {X 0,Y 307.348,Z 423.022,A -85,B 0,C 180,E1 -16496.397,E2 -16496.397} C_VEL
LIN {X 0,Y 308.919,Z 413.748,A -85,B 0,C 180,E1 -16497.983,E2 -16497.983} C_VEL
LIN {X 0,Y 310.501,Z 404.099,A -85,B 0,C 180,E1 -16499.306,E2 -16499.306} C_VEL
LIN {X 0,Y 311.871,Z 393.64,A -85,B 0,C 180,E1 -16500.467,E2 -16500.467} C_VEL
LIN {X 0,Y 313.032,Z 382.36,A -85,B 0,C 180,E1 -16501.443,E2 -16501.443} C_VEL
LIN {X 0,Y 313.838,Z 369.557,A -85,B 0,C 180,E1 -16502.276,E2 -16502.276} C_VEL
LIN {X 0,Y 314.327,Z 356.519,A -85,B 0,C 180,E1 -16502.848,E2 -16502.848} C_VEL
LIN {X 0,Y 315.288,Z 314.203,A -85,B 0,C 180,E1 -16503.867,E2 -16503.867} C_VEL
LIN {X 0,Y 315.607,Z 301.776,A -85,B 0,C 180,E1 -16504.155,E2 -16504.155} C_VEL
LIN {X 0,Y 306.347,Z 283.316,A -85,B 0,C 180,E1 -16505.667,E2 -16505.667} C_VEL
LIN {X 0,Y 299.695,Z 271.506,A -85,B 0,C 180,E1 -16506.786,E2 -16506.786} C_VEL
LIN {X 0,Y 298.519,Z 268.901,A -85,B 0,C 180,E1 -16507.082,E2 -16507.082} C_VEL
LIN {X 0,Y 298.416,Z 268.346,A -85,B 0,C 180,E1 -16507.354,E2 -16507.354} C_VEL
LIN {X 0,Y 298.347,Z 268.309,A -85,B 0,C 180,E1 -16511.268,E2 -16511.268} C_VEL
LIN {X 0,Y 298.355,Z 268.317,A -85,B 0,C 180,E1 -16515.034,E2 -16515.034} C_VEL
LIN {X 0,Y 298.347,Z 268.32,A -85,B 0,C 180,E1 -16518.921,E2 -16518.921} C_VEL
LIN {X 0,Y 298.385,Z 268.288,A -85,B 0,C 180,E1 -16522.237,E2 -16522.237} C_VEL
LIN {X 0,Y 298.403,Z 268.294,A -85,B 0,C 180,E1 -16523.761,E2 -16523.761} C_VEL
LIN {X 0,Y 297.722,Z 268.396,A -85,B 0,C 180,E1 -16524.888,E2 -16524.888} C_VEL
LIN {X 0,Y 294.83,Z 268.758,A -85,B 0,C 180,E1 -16526.723,E2 -16526.723} C_VEL
LIN {X 0,Y 292.397,Z 269.038,A -85,B 0,C 180,E1 -16528.212,E2 -16528.212} C_VEL
LIN {X 0,Y 291.377,Z 269.151,A -85,B 0,C 180,E1 -16529.366,E2 -16529.366} C_VEL
LIN {X 0,Y 291.307,Z 269.159,A -85,B 0,C 180,E1 -16529.757,E2 -16529.757} C_VEL
LIN {X 0,Y 291.348,Z 269.195,A -85,B 0,C 180,E1 -16533.191,E2 -16533.191} C_VEL
LIN {X 0,Y 291.363,Z 269.145,A -85,B 0,C 180,E1 -16537.298,E2 -16537.298} C_VEL
LIN {X 0,Y 291.456,Z 269.152,A -85,B 0,C 180,E1 -16540.27,E2 -16540.27} C_VEL
LIN {X 0,Y 291.538,Z 269.16,A -85,B 0,C 180,E1 -16544.634,E2 -16544.634} C_VEL
LIN {X 0,Y 291.525,Z 269.169,A -85,B 0,C 180,E1 -16548.88,E2 -16548.88} C_VEL
LIN {X 0,Y 291.646,Z 269.144,A -85,B 0,C 180,E1 -16551.686,E2 -16551.686} C_VEL
LIN {X 0,Y 291.59,Z 269.159,A -85,B 0,C 180,E1 -16554.467,E2 -16554.467} C_VEL
LIN {X 0,Y 291.874,Z 269.127,A -85,B 0,C 180,E1 -16558.62,E2 -16558.62} C_VEL
LIN {X 0,Y 291.866,Z 269.115,A -85,B 0,C 180,E1 -16561.379,E2 -16561.379} C_VEL
LIN {X 0,Y 291.679,Z 269.139,A -85,B 0,C 180,E1 -16566.919,E2 -16566.919} C_VEL
LIN {X 0,Y 291.564,Z 269.166,A -85,B 0,C 180,E1 -16569.714,E2 -16569.714} C_VEL
LIN {X 0,Y 291.51,Z 269.162,A -85,B 0,C 180,E1 -16573.951,E2 -16573.951} C_VEL
LIN {X 0,Y 291.437,Z 269.181,A -85,B 0,C 180,E1 -16576.821,E2 -16576.821} C_VEL
LIN {X 0,Y 291.421,Z 269.185,A -85,B 0,C 180,E1 -16579.86,E2 -16579.86} C_VEL
LIN {X 0,Y 291.355,Z 269.193,A -85,B 0,C 180,E1 -16584.209,E2 -16584.209} C_VEL
LIN {X 0,Y 291.327,Z 269.168,A -85,B 0,C 180,E1 -16587.281,E2 -16587.281} C_VEL
LIN {X 0,Y 291.297,Z 269.199,A -85,B 0,C 180,E1 -16590.441,E2 -16590.441} C_VEL
LIN {X 0,Y 291.34,Z 269.172,A -85,B 0,C 180,E1 -16593.699,E2 -16593.699} C_VEL
LIN {X 0,Y 291.35,Z 269.19,A -85,B 0,C 180,E1 -16597.248,E2 -16597.248} C_VEL
LIN {X 0,Y 291.297,Z 269.201,A -85,B 0,C 180,E1 -16600.648,E2 -16600.648} C_VEL
LIN {X 0,Y 291.279,Z 269.199,A -85,B 0,C 180,E1 -16604.404,E2 -16604.404} C_VEL
LIN {X 0,Y 291.292,Z 269.198,A -85,B 0,C 180,E1 -16608.412,E2 -16608.412} C_VEL
LIN {X 0,Y 291.348,Z 269.452,A -85,B 0,C 180,E1 -16609.152,E2 -16609.152} C_VEL
LIN {X 0,Y 294.082,Z 278.883,A -85,B 0,C 180,E1 -16612.058,E2 -16612.058} C_VEL
LIN {X 0,Y 296.77,Z 289.18,A -85,B 0,C 180,E1 -16615.001,E2 -16615.001} C_VEL
LIN {X 0,Y 299.275,Z 300.815,A -85,B 0,C 180,E1 -16618.102,E2 -16618.102} C_VEL
LIN {X 0,Y 299.585,Z 304.164,A -85,B 0,C 180,E1 -16618.929,E2 -16618.929} C_VEL
LIN {X 0,Y 298.573,Z 311.467,A -85,B 0,C 180,E1 -16620.527,E2 -16620.527} C_VEL
LIN {X 0,Y 299.421,Z 317.232,A -85,B 0,C 180,E1 -16620.852,E2 -16620.852} C_VEL
LIN {X 0,Y 303.948,Z 345.691,A -85,B 0,C 180,E1 -16622.143,E2 -16622.143} C_VEL
LIN {X 0,Y 307.001,Z 370.794,A -85,B 0,C 180,E1 -16623.137,E2 -16623.137} C_VEL
LIN {X 0,Y 307.383,Z 378.108,A -85,B 0,C 180,E1 -16623.369,E2 -16623.369} C_VEL
LIN {X 0,Y 305.934,Z 423.25,A -85,B 0,C 180,E1 -16624.441,E2 -16624.441} C_VEL
LIN {X 0,Y 304.996,Z 436.442,A -85,B 0,C 180,E1 -16624.995,E2 -16624.995} C_VEL
LIN {X 0,Y 303.411,Z 449.729,A -85,B 0,C 180,E1 -16625.814,E2 -16625.814} C_VEL
LIN {X 0,Y 301.397,Z 461.711,A -85,B 0,C 180,E1 -16626.828,E2 -16626.828} C_VEL
LIN {X 0,Y 299.222,Z 473.212,A -85,B 0,C 180,E1 -16628.107,E2 -16628.107} C_VEL
LIN {X 0,Y 297.175,Z 483.625,A -85,B 0,C 180,E1 -16629.584,E2 -16629.584} C_VEL
LIN {X 0,Y 295.118,Z 493.026,A -85,B 0,C 180,E1 -16631.247,E2 -16631.247} C_VEL
LIN {X 0,Y 293.25,Z 502.193,A -85,B 0,C 180,E1 -16633.286,E2 -16633.286} C_VEL
LIN {X 0,Y 291.847,Z 509.641,A -85,B 0,C 180,E1 -16635.353,E2 -16635.353} C_VEL
LIN {X 0,Y 290.786,Z 515.661,A -85,B 0,C 180,E1 -16637.436,E2 -16637.436} C_VEL
LIN {X 0,Y 290.101,Z 520.458,A -85,B 0,C 180,E1 -16639.531,E2 -16639.531} C_VEL
LIN {X 0,Y 289.939,Z 524.183,A -85,B 0,C 180,E1 -16641.637,E2 -16641.637} C_VEL
LIN {X 0,Y 290.046,Z 526.578,A -85,B 0,C 180,E1 -16643.443,E2 -16643.443} C_VEL
LIN {X 0,Y 290.316,Z 528.695,A -85,B 0,C 180,E1 -16645.835,E2 -16645.835} C_VEL
LIN {X 0,Y 290.561,Z 529.387,A -85,B 0,C 180,E1 -16647.227,E2 -16647.227} C_VEL
LIN {X 0,Y 290.572,Z 529.633,A -85,B 0,C 180,E1 -16648.614,E2 -16648.614} C_VEL
LIN {X 0,Y 290.698,Z 529.45,A -85,B 0,C 180,E1 -16649.999,E2 -16649.999} C_VEL
LIN {X 0,Y 290.631,Z 528.84,A -85,B 0,C 180,E1 -16651.385,E2 -16651.385} C_VEL
LIN {X 0,Y 290.633,Z 527.83,A -85,B 0,C 180,E1 -16652.771,E2 -16652.771} C_VEL
LIN {X 0,Y 290.486,Z 526.362,A -85,B 0,C 180,E1 -16654.162,E2 -16654.162} C_VEL
LIN {X 0,Y 290.19,Z 522.283,A -85,B 0,C 180,E1 -16656.8,E2 -16656.8} C_VEL
LIN {X 0,Y 290.108,Z 517.441,A -85,B 0,C 180,E1 -16659.059,E2 -16659.059} C_VEL
LIN {X 0,Y 290.349,Z 511.663,A -85,B 0,C 180,E1 -16661.165,E2 -16661.165} C_VEL
LIN {X 0,Y 290.966,Z 504.458,A -85,B 0,C 180,E1 -16663.265,E2 -16663.265} C_VEL
LIN {X 0,Y 291.713,Z 497.112,A -85,B 0,C 180,E1 -16665.009,E2 -16665.009} C_VEL
LIN {X 0,Y 293.115,Z 487.274,A -85,B 0,C 180,E1 -16666.9,E2 -16666.9} C_VEL
LIN {X 0,Y 294.236,Z 478.563,A -85,B 0,C 180,E1 -16668.269,E2 -16668.269} C_VEL
LIN {X 0,Y 295.575,Z 467.988,A -85,B 0,C 180,E1 -16669.624,E2 -16669.624} C_VEL
LIN {X 0,Y 297.067,Z 456.412,A -85,B 0,C 180,E1 -16670.784,E2 -16670.784} C_VEL
LIN {X 0,Y 298.298,Z 444.406,A -85,B 0,C 180,E1 -16671.69,E2 -16671.69} C_VEL
LIN {X 0,Y 299.22,Z 431.412,A -85,B 0,C 180,E1 -16672.391,E2 -16672.391} C_VEL
LIN {X 0,Y 299.764,Z 419.324,A -85,B 0,C 180,E1 -16672.803,E2 -16672.803} C_VEL
LIN {X 0,Y 300.573,Z 373.108,A -85,B 0,C 180,E1 -16673.903,E2 -16673.903} C_VEL
LIN {X 0,Y 296.214,Z 327.903,A -85,B 0,C 180,E1 -16675.358,E2 -16675.358} C_VEL
LIN {X 0,Y 294.527,Z 313.734,A -85,B 0,C 180,E1 -16675.862,E2 -16675.862} C_VEL
LIN {X 0,Y 295.877,Z 301.877,A -85,B 0,C 180,E1 -16678.362,E2 -16678.362} C_VEL
LIN {X 0,Y 296.628,Z 295.082,A -85,B 0,C 180,E1 -16679.837,E2 -16679.837} C_VEL
LIN {X 0,Y 295.987,Z 290.328,A -85,B 0,C 180,E1 -16680.955,E2 -16680.955} C_VEL
LIN {X 0,Y 293.575,Z 278.712,A -85,B 0,C 180,E1 -16683.819,E2 -16683.819} C_VEL
LIN {X 0,Y 291.412,Z 269.301,A -85,B 0,C 180,E1 -16686.297,E2 -16686.297} C_VEL
LIN {X 0,Y 291.294,Z 269.194,A -85,B 0,C 180,E1 -16690.647,E2 -16690.647} C_VEL
LIN {X 0,Y 291.275,Z 269.186,A -85,B 0,C 180,E1 -16694.403,E2 -16694.403} C_VEL
LIN {X 0,Y 291.287,Z 269.199,A -85,B 0,C 180,E1 -16698.411,E2 -16698.411} C_VEL
LIN {X 0,Y 291.326,Z 269.191,A -85,B 0,C 180,E1 -16701.154,E2 -16701.154} C_VEL
LIN {X 0,Y 291.347,Z 269.193,A -85,B 0,C 180,E1 -16704.624,E2 -16704.624} C_VEL
LIN {X 0,Y 291.355,Z 269.182,A -85,B 0,C 180,E1 -16707.949,E2 -16707.949} C_VEL
LIN {X 0,Y 291.313,Z 269.199,A -85,B 0,C 180,E1 -16711.151,E2 -16711.151} C_VEL
LIN {X 0,Y 291.348,Z 269.187,A -85,B 0,C 180,E1 -16714.266,E2 -16714.266} C_VEL
LIN {X 0,Y 291.354,Z 269.192,A -85,B 0,C 180,E1 -16717.297,E2 -16717.297} C_VEL
LIN {X 0,Y 291.381,Z 269.186,A -85,B 0,C 180,E1 -16720.265,E2 -16720.265} C_VEL
LIN {X 0,Y 291.488,Z 269.175,A -85,B 0,C 180,E1 -16724.665,E2 -16724.665} C_VEL
LIN {X 0,Y 291.518,Z 269.165,A -85,B 0,C 180,E1 -16728.88,E2 -16728.88} C_VEL
LIN {X 0,Y 291.639,Z 269.149,A -85,B 0,C 180,E1 -16731.687,E2 -16731.687} C_VEL
LIN {X 0,Y 291.586,Z 269.165,A -85,B 0,C 180,E1 -16734.468,E2 -16734.468} C_VEL
LIN {X 0,Y 291.86,Z 269.12,A -85,B 0,C 180,E1 -16738.62,E2 -16738.62} C_VEL
LIN {X 0,Y 291.866,Z 269.123,A -85,B 0,C 180,E1 -16741.38,E2 -16741.38} C_VEL
LIN {X 0,Y 291.672,Z 269.145,A -85,B 0,C 180,E1 -16746.92,E2 -16746.92} C_VEL
LIN {X 0,Y 291.553,Z 269.157,A -85,B 0,C 180,E1 -16749.715,E2 -16749.715} C_VEL
LIN {X 0,Y 291.505,Z 269.173,A -85,B 0,C 180,E1 -16753.951,E2 -16753.951} C_VEL
LIN {X 0,Y 291.419,Z 269.173,A -85,B 0,C 180,E1 -16756.822,E2 -16756.822} C_VEL
LIN {X 0,Y 291.383,Z 269.184,A -85,B 0,C 180,E1 -16759.843,E2 -16759.843} C_VEL
LIN {X 0,Y 291.325,Z 269.192,A -85,B 0,C 180,E1 -16764.212,E2 -16764.212} C_VEL
LIN {X 0,Y 291.32,Z 269.189,A -85,B 0,C 180,E1 -16767.282,E2 -16767.282} C_VEL
LIN {X 0,Y 291.294,Z 269.199,A -85,B 0,C 180,E1 -16770.442,E2 -16770.442} C_VEL
LIN {X 0,Y 291.337,Z 269.188,A -85,B 0,C 180,E1 -16773.7,E2 -16773.7} C_VEL
LIN {X 0,Y 291.346,Z 269.192,A -85,B 0,C 180,E1 -16777.249,E2 -16777.249} C_VEL
LIN {X 0,Y 291.294,Z 269.187,A -85,B 0,C 180,E1 -16780.65,E2 -16780.65} C_VEL
LIN {X 0,Y 291.277,Z 269.185,A -85,B 0,C 180,E1 -16784.405,E2 -16784.405} C_VEL
LIN {X 0,Y 291.29,Z 269.199,A -85,B 0,C 180,E1 -16788.413,E2 -16788.413} C_VEL
LIN {X 0,Y 291.33,Z 269.188,A -85,B 0,C 180,E1 -16791.157,E2 -16791.157} C_VEL
LIN {X 0,Y 291.352,Z 269.186,A -85,B 0,C 180,E1 -16794.626,E2 -16794.626} C_VEL
LIN {X 0,Y 291.362,Z 269.187,A -85,B 0,C 180,E1 -16797.951,E2 -16797.951} C_VEL
LIN {X 0,Y 291.312,Z 269.191,A -85,B 0,C 180,E1 -16801.152,E2 -16801.152} C_VEL
LIN {X 0,Y 291.345,Z 269.187,A -85,B 0,C 180,E1 -16804.266,E2 -16804.266} C_VEL
LIN {X 0,Y 291.35,Z 269.196,A -85,B 0,C 180,E1 -16807.298,E2 -16807.298} C_VEL
LIN {X 0,Y 291.385,Z 269.155,A -85,B 0,C 180,E1 -16810.266,E2 -16810.266} C_VEL
LIN {X 0,Y 291.391,Z 269.298,A -85,B 0,C 180,E1 -16812.3,E2 -16812.3} C_VEL
LIN {X 0,Y 291.582,Z 270.207,A -85,B 0,C 180,E1 -16812.548,E2 -16812.548} C_VEL
LIN {X 0,Y 299.874,Z 289.331,A -85,B 0,C 180,E1 -16813.729,E2 -16813.729} C_VEL
LIN {X 0,Y 302.17,Z 295.8,A -85,B 0,C 180,E1 -16814.067,E2 -16814.067} C_VEL
LIN {X 0,Y 300.973,Z 355.721,A -85,B 0,C 180,E1 -16815.506,E2 -16815.506} C_VEL
LIN {X 0,Y 300.606,Z 368.353,A -85,B 0,C 180,E1 -16816.049,E2 -16816.049} C_VEL
LIN {X 0,Y 300.084,Z 381.177,A -85,B 0,C 180,E1 -16816.887,E2 -16816.887} C_VEL
LIN {X 0,Y 299.147,Z 393.454,A -85,B 0,C 180,E1 -16817.966,E2 -16817.966} C_VEL
LIN {X 0,Y 297.951,Z 404.979,A -85,B 0,C 180,E1 -16819.296,E2 -16819.296} C_VEL
LIN {X 0,Y 296.842,Z 415.302,A -85,B 0,C 180,E1 -16820.805,E2 -16820.805} C_VEL
LIN {X 0,Y 295.697,Z 424.628,A -85,B 0,C 180,E1 -16822.489,E2 -16822.489} C_VEL
LIN {X 0,Y 294.421,Z 433.62,A -85,B 0,C 180,E1 -16824.522,E2 -16824.522} C_VEL
LIN {X 0,Y 293.316,Z 440.877,A -85,B 0,C 180,E1 -16826.567,E2 -16826.567} C_VEL
LIN {X 0,Y 292.486,Z 446.694,A -85,B 0,C 180,E1 -16828.624,E2 -16828.624} C_VEL
LIN {X 0,Y 291.896,Z 451.289,A -85,B 0,C 180,E1 -16830.69,E2 -16830.69} C_VEL
LIN {X 0,Y 291.32,Z 454.831,A -85,B 0,C 180,E1 -16832.766,E2 -16832.766} C_VEL
LIN {X 0,Y 291.198,Z 456.629,A -85,B 0,C 180,E1 -16834.153,E2 -16834.153} C_VEL
LIN {X 0,Y 291.19,Z 457.978,A -85,B 0,C 180,E1 -16835.541,E2 -16835.541} C_VEL
LIN {X 0,Y 291.173,Z 459.565,A -85,B 0,C 180,E1 -16838.327,E2 -16838.327} C_VEL
LIN {X 0,Y 291.275,Z 459.762,A -85,B 0,C 180,E1 -16839.724,E2 -16839.724} C_VEL
LIN {X 0,Y 291.701,Z 458.958,A -85,B 0,C 180,E1 -16842.524,E2 -16842.524} C_VEL
LIN {X 0,Y 292.075,Z 457.979,A -85,B 0,C 180,E1 -16843.924,E2 -16843.924} C_VEL
LIN {X 0,Y 293.052,Z 455.155,A -85,B 0,C 180,E1 -16846.404,E2 -16846.404} C_VEL
LIN {X 0,Y 294.21,Z 451.056,A -85,B 0,C 180,E1 -16848.813,E2 -16848.813} C_VEL
LIN {X 0,Y 295.491,Z 446.275,A -85,B 0,C 180,E1 -16850.902,E2 -16850.902} C_VEL
LIN {X 0,Y 297.103,Z 440.192,A -85,B 0,C 180,E1 -16852.973,E2 -16852.973} C_VEL
LIN {X 0,Y 298.896,Z 432.543,A -85,B 0,C 180,E1 -16855.039,E2 -16855.039} C_VEL
LIN {X 0,Y 300.865,Z 423.555,A -85,B 0,C 180,E1 -16856.95,E2 -16856.95} C_VEL
LIN {X 0,Y 302.619,Z 413.86,A -85,B 0,C 180,E1 -16858.62,E2 -16858.62} C_VEL
LIN {X 0,Y 304.384,Z 402.618,A -85,B 0,C 180,E1 -16860.145,E2 -16860.145} C_VEL
LIN {X 0,Y 305.909,Z 391.5,A -85,B 0,C 180,E1 -16861.318,E2 -16861.318} C_VEL
LIN {X 0,Y 307.036,Z 380.219,A -85,B 0,C 180,E1 -16862.249,E2 -16862.249} C_VEL
LIN {X 0,Y 307.791,Z 367.428,A -85,B 0,C 180,E1 -16863.035,E2 -16863.035} C_VEL
LIN {X 0,Y 308.201,Z 354.597,A -85,B 0,C 180,E1 -16863.542,E2 -16863.542} C_VEL
LIN {X 0,Y 309.172,Z 313.898,A -85,B 0,C 180,E1 -16864.528,E2 -16864.528} C_VEL
LIN {X 0,Y 309.48,Z 304.059,A -85,B 0,C 180,E1 -16864.756,E2 -16864.756} C_VEL
LIN {X 0,Y 301.229,Z 287.524,A -85,B 0,C 180,E1 -16866.153,E2 -16866.153} C_VEL
LIN {X 0,Y 294.328,Z 275.26,A -85,B 0,C 180,E1 -16867.354,E2 -16867.354} C_VEL
LIN {X 0,Y 292.565,Z 272.334,A -85,B 0,C 180,E1 -16867.667,E2 -16867.667} C_VEL
LIN {X 0,Y 291.436,Z 269.754,A -85,B 0,C 180,E1 -16867.977,E2 -16867.977} C_VEL
LIN {X 0,Y 291.337,Z 269.259,A -85,B 0,C 180,E1 -16868.207,E2 -16868.207} C_VEL
LIN {X 0,Y 291.294,Z 269.185,A -85,B 0,C 180,E1 -16871.588,E2 -16871.588} C_VEL
LIN {X 0,Y 291.281,Z 269.188,A -85,B 0,C 180,E1 -16875.596,E2 -16875.596} C_VEL
LIN {X 0,Y 291.299,Z 269.2,A -85,B 0,C 180,E1 -16879.351,E2 -16879.351} C_VEL
LIN {X 0,Y 291.384,Z 269.159,A -85,B 0,C 180,E1 -16882.915,E2 -16882.915} C_VEL
LIN {X 0,Y 291.342,Z 269.196,A -85,B 0,C 180,E1 -16886.301,E2 -16886.301} C_VEL
LIN {X 0,Y 291.307,Z 269.159,A -85,B 0,C 180,E1 -16889.757,E2 -16889.757} C_VEL
LIN {X 0,Y 290.669,Z 269.249,A -85,B 0,C 180,E1 -16890.912,E2 -16890.912} C_VEL
LIN {X 0,Y 287.814,Z 269.633,A -85,B 0,C 180,E1 -16892.792,E2 -16892.792} C_VEL
LIN {X 0,Y 285.391,Z 269.935,A -85,B 0,C 180,E1 -16894.319,E2 -16894.319} C_VEL
LIN {X 0,Y 284.375,Z 270.045,A -85,B 0,C 180,E1 -16895.502,E2 -16895.502} C_VEL
LIN {X 0,Y 284.307,Z 270.045,A -85,B 0,C 180,E1 -16895.902,E2 -16895.902} C_VEL
LIN {X 0,Y 284.386,Z 270.025,A -85,B 0,C 180,E1 -16899.898,E2 -16899.898} C_VEL
LIN {X 0,Y 284.476,Z 270.04,A -85,B 0,C 180,E1 -16904.469,E2 -16904.469} C_VEL
LIN {X 0,Y 284.479,Z 270.047,A -85,B 0,C 180,E1 -16908.601,E2 -16908.601} C_VEL
LIN {X 0,Y 284.604,Z 270.019,A -85,B 0,C 180,E1 -16911.479,E2 -16911.479} C_VEL
LIN {X 0,Y 284.561,Z 270.035,A -85,B 0,C 180,E1 -16914.33,E2 -16914.33} C_VEL
LIN {X 0,Y 284.84,Z 270.003,A -85,B 0,C 180,E1 -16918.586,E2 -16918.586} C_VEL
LIN {X 0,Y 284.833,Z 269.99,A -85,B 0,C 180,E1 -16921.414,E2 -16921.414} C_VEL
LIN {X 0,Y 284.635,Z 270.015,A -85,B 0,C 180,E1 -16927.091,E2 -16927.091} C_VEL
LIN {X 0,Y 284.51,Z 270.045,A -85,B 0,C 180,E1 -16929.957,E2 -16929.957} C_VEL
LIN {X 0,Y 284.459,Z 270.044,A -85,B 0,C 180,E1 -16934.304,E2 -16934.304} C_VEL
LIN {X 0,Y 284.378,Z 270.055,A -85,B 0,C 180,E1 -16938.74,E2 -16938.74} C_VEL
LIN {X 0,Y 284.306,Z 270.063,A -85,B 0,C 180,E1 -16941.765,E2 -16941.765} C_VEL
LIN {X 0,Y 284.301,Z 270.069,A -85,B 0,C 180,E1 -16944.85,E2 -16944.85} C_VEL
LIN {X 0,Y 284.257,Z 270.049,A -85,B 0,C 180,E1 -16948.018,E2 -16948.018} C_VEL
LIN {X 0,Y 284.273,Z 270.074,A -85,B 0,C 180,E1 -16951.277,E2 -16951.277} C_VEL
LIN {X 0,Y 284.334,Z 270.058,A -85,B 0,C 180,E1 -16955.347,E2 -16955.347} C_VEL
LIN {X 0,Y 284.292,Z 270.059,A -85,B 0,C 180,E1 -16958.172,E2 -16958.172} C_VEL
LIN {X 0,Y 284.234,Z 270.074,A -85,B 0,C 180,E1 -16962.117,E2 -16962.117} C_VEL
LIN {X 0,Y 284.235,Z 270.071,A -85,B 0,C 180,E1 -16966.186,E2 -16966.186} C_VEL
LIN {X 0,Y 284.278,Z 270.273,A -85,B 0,C 180,E1 -16968.307,E2 -16968.307} C_VEL
LIN {X 0,Y 287.23,Z 280.355,A -85,B 0,C 180,E1 -16971.534,E2 -16971.534} C_VEL
LIN {X 0,Y 289.794,Z 290.067,A -85,B 0,C 180,E1 -16974.406,E2 -16974.406} C_VEL
LIN {X 0,Y 292.133,Z 300.747,A -85,B 0,C 180,E1 -16977.353,E2 -16977.353} C_VEL
LIN {X 0,Y 292.838,Z 305.275,A -85,B 0,C 180,E1 -16978.534,E2 -16978.534} C_VEL
LIN {X 0,Y 292.144,Z 310.732,A -85,B 0,C 180,E1 -16979.737,E2 -16979.737} C_VEL
LIN {X 0,Y 297.071,Z 341.385,A -85,B 0,C 180,E1 -16981.247,E2 -16981.247} C_VEL
LIN {X 0,Y 300.276,Z 366.367,A -85,B 0,C 180,E1 -16982.297,E2 -16982.297} C_VEL
LIN {X 0,Y 301.202,Z 377.86,A -85,B 0,C 180,E1 -16982.71,E2 -16982.71} C_VEL
LIN {X 0,Y 299.662,Z 423.295,A -85,B 0,C 180,E1 -16983.819,E2 -16983.819} C_VEL
LIN {X 0,Y 298.594,Z 436.943,A -85,B 0,C 180,E1 -16984.421,E2 -16984.421} C_VEL
LIN {X 0,Y 296.961,Z 449.792,A -85,B 0,C 180,E1 -16985.254,E2 -16985.254} C_VEL
LIN {X 0,Y 294.874,Z 461.554,A -85,B 0,C 180,E1 -16986.284,E2 -16986.284} C_VEL
LIN {X 0,Y 292.645,Z 472.926,A -85,B 0,C 180,E1 -16987.589,E2 -16987.589} C_VEL
LIN {X 0,Y 290.518,Z 483.229,A -85,B 0,C 180,E1 -16989.095,E2 -16989.095} C_VEL
LIN {X 0,Y 288.383,Z 492.526,A -85,B 0,C 180,E1 -16990.792,E2 -16990.792} C_VEL
LIN {X 0,Y 286.391,Z 501.629,A -85,B 0,C 180,E1 -16992.874,E2 -16992.874} C_VEL
LIN {X 0,Y 284.964,Z 509.028,A -85,B 0,C 180,E1 -16994.991,E2 -16994.991} C_VEL
LIN {X 0,Y 283.795,Z 514.993,A -85,B 0,C 180,E1 -16997.121,E2 -16997.121} C_VEL
LIN {X 0,Y 283.064,Z 519.748,A -85,B 0,C 180,E1 -16999.268,E2 -16999.268} C_VEL
LIN {X 0,Y 282.867,Z 523.438,A -85,B 0,C 180,E1 -17001.426,E2 -17001.426} C_VEL
LIN {X 0,Y 282.984,Z 525.955,A -85,B 0,C 180,E1 -17003.42,E2 -17003.42} C_VEL
LIN {X 0,Y 283.239,Z 527.882,A -85,B 0,C 180,E1 -17005.731,E2 -17005.731} C_VEL
LIN {X 0,Y 283.489,Z 528.56,A -85,B 0,C 180,E1 -17007.157,E2 -17007.157} C_VEL
LIN {X 0,Y 283.524,Z 528.774,A -85,B 0,C 180,E1 -17008.579,E2 -17008.579} C_VEL
LIN {X 0,Y 283.649,Z 528.575,A -85,B 0,C 180,E1 -17009.999,E2 -17009.999} C_VEL
LIN {X 0,Y 283.58,Z 527.947,A -85,B 0,C 180,E1 -17011.419,E2 -17011.419} C_VEL
LIN {X 0,Y 283.584,Z 526.92,A -85,B 0,C 180,E1 -17012.84,E2 -17012.84} C_VEL
LIN {X 0,Y 283.42,Z 525.413,A -85,B 0,C 180,E1 -17014.266,E2 -17014.266} C_VEL
LIN {X 0,Y 283.14,Z 521.514,A -85,B 0,C 180,E1 -17016.847,E2 -17016.847} C_VEL
LIN {X 0,Y 283.046,Z 516.404,A -85,B 0,C 180,E1 -17019.287,E2 -17019.287} C_VEL
LIN {X 0,Y 283.426,Z 509.458,A -85,B 0,C 180,E1 -17021.804,E2 -17021.804} C_VEL
LIN {X 0,Y 284.119,Z 501.899,A -85,B 0,C 180,E1 -17023.955,E2 -17023.955} C_VEL
LIN {X 0,Y 285.21,Z 493.234,A -85,B 0,C 180,E1 -17025.946,E2 -17025.946} C_VEL
LIN {X 0,Y 286.426,Z 483.928,A -85,B 0,C 180,E1 -17027.676,E2 -17027.676} C_VEL
LIN {X 0,Y 287.912,Z 473.419,A -85,B 0,C 180,E1 -17029.24,E2 -17029.24} C_VEL
LIN {X 0,Y 289.305,Z 463.387,A -85,B 0,C 180,E1 -17030.438,E2 -17030.438} C_VEL
LIN {X 0,Y 290.835,Z 450.654,A -85,B 0,C 180,E1 -17031.623,E2 -17031.623} C_VEL
LIN {X 0,Y 292.018,Z 438.241,A -85,B 0,C 180,E1 -17032.46,E2 -17032.46} C_VEL
LIN {X 0,Y 292.793,Z 425.315,A -85,B 0,C 180,E1 -17033.059,E2 -17033.059} C_VEL
LIN {X 0,Y 293.412,Z 400.844,A -85,B 0,C 180,E1 -17033.7,E2 -17033.7} C_VEL
LIN {X 0,Y 293.907,Z 373.68,A -85,B 0,C 180,E1 -17034.359,E2 -17034.359} C_VEL
LIN {X 0,Y 289.591,Z 328.726,A -85,B 0,C 180,E1 -17035.844,E2 -17035.844} C_VEL
LIN {X 0,Y 287.757,Z 312.809,A -85,B 0,C 180,E1 -17036.429,E2 -17036.429} C_VEL
LIN {X 0,Y 289.608,Z 297.203,A -85,B 0,C 180,E1 -17039.832,E2 -17039.832} C_VEL
LIN {X 0,Y 289.441,Z 293.685,A -85,B 0,C 180,E1 -17040.656,E2 -17040.656} C_VEL
LIN {X 0,Y 286.867,Z 280.976,A -85,B 0,C 180,E1 -17043.853,E2 -17043.853} C_VEL
LIN {X 0,Y 284.379,Z 270.168,A -85,B 0,C 180,E1 -17046.763,E2 -17046.763} C_VEL
LIN {X 0,Y 284.276,Z 270.062,A -85,B 0,C 180,E1 -17049.998,E2 -17049.998} C_VEL
LIN {X 0,Y 284.227,Z 270.064,A -85,B 0,C 180,E1 -17054.187,E2 -17054.187} C_VEL
LIN {X 0,Y 284.232,Z 270.078,A -85,B 0,C 180,E1 -17058.117,E2 -17058.117} C_VEL
LIN {X 0,Y 284.3,Z 270.065,A -85,B 0,C 180,E1 -17062.281,E2 -17062.281} C_VEL
LIN {X 0,Y 284.299,Z 270.069,A -85,B 0,C 180,E1 -17065.35,E2 -17065.35} C_VEL
LIN {X 0,Y 284.269,Z 270.066,A -85,B 0,C 180,E1 -17068.723,E2 -17068.723} C_VEL
LIN {X 0,Y 284.318,Z 270.068,A -85,B 0,C 180,E1 -17072.854,E2 -17072.854} C_VEL
LIN {X 0,Y 284.318,Z 270.066,A -85,B 0,C 180,E1 -17076.703,E2 -17076.703} C_VEL
LIN {X 0,Y 284.322,Z 270.059,A -85,B 0,C 180,E1 -17081.256,E2 -17081.256} C_VEL
LIN {X 0,Y 284.453,Z 270.05,A -85,B 0,C 180,E1 -17085.696,E2 -17085.696} C_VEL
LIN {X 0,Y 284.504,Z 270.036,A -85,B 0,C 180,E1 -17090.043,E2 -17090.043} C_VEL
LIN {X 0,Y 284.629,Z 270.03,A -85,B 0,C 180,E1 -17092.909,E2 -17092.909} C_VEL
LIN {X 0,Y 284.827,Z 269.995,A -85,B 0,C 180,E1 -17098.586,E2 -17098.586} C_VEL
LIN {X 0,Y 284.832,Z 269.999,A -85,B 0,C 180,E1 -17101.414,E2 -17101.414} C_VEL
LIN {X 0,Y 284.625,Z 270.021,A -85,B 0,C 180,E1 -17107.092,E2 -17107.092} C_VEL
LIN {X 0,Y 284.501,Z 270.036,A -85,B 0,C 180,E1 -17109.958,E2 -17109.958} C_VEL
LIN {X 0,Y 284.454,Z 270.051,A -85,B 0,C 180,E1 -17114.305,E2 -17114.305} C_VEL
LIN {X 0,Y 284.323,Z 270.062,A -85,B 0,C 180,E1 -17118.744,E2 -17118.744} C_VEL
LIN {X 0,Y 284.302,Z 270.068,A -85,B 0,C 180,E1 -17123.299,E2 -17123.299} C_VEL
LIN {X 0,Y 284.278,Z 270.066,A -85,B 0,C 180,E1 -17127.13,E2 -17127.13} C_VEL
LIN {X 0,Y 284.266,Z 270.077,A -85,B 0,C 180,E1 -17130.085,E2 -17130.085} C_VEL
LIN {X 0,Y 284.298,Z 270.063,A -85,B 0,C 180,E1 -17132.947,E2 -17132.947} C_VEL
LIN {X 0,Y 284.312,Z 270.069,A -85,B 0,C 180,E1 -17136.39,E2 -17136.39} C_VEL
LIN {X 0,Y 284.277,Z 270.064,A -85,B 0,C 180,E1 -17140,E2 -17140} C_VEL
LIN {X 0,Y 284.228,Z 270.057,A -85,B 0,C 180,E1 -17144.189,E2 -17144.189} C_VEL
LIN {X 0,Y 284.235,Z 270.08,A -85,B 0,C 180,E1 -17148.12,E2 -17148.12} C_VEL
LIN {X 0,Y 284.292,Z 270.054,A -85,B 0,C 180,E1 -17151.83,E2 -17151.83} C_VEL
LIN {X 0,Y 284.305,Z 270.067,A -85,B 0,C 180,E1 -17155.352,E2 -17155.352} C_VEL
LIN {X 0,Y 284.275,Z 270.068,A -85,B 0,C 180,E1 -17158.725,E2 -17158.725} C_VEL
LIN {X 0,Y 284.258,Z 270.077,A -85,B 0,C 180,E1 -17161.983,E2 -17161.983} C_VEL
LIN {X 0,Y 284.288,Z 270.063,A -85,B 0,C 180,E1 -17165.15,E2 -17165.15} C_VEL
LIN {X 0,Y 284.297,Z 270.067,A -85,B 0,C 180,E1 -17168.236,E2 -17168.236} C_VEL
LIN {X 0,Y 284.362,Z 270.209,A -85,B 0,C 180,E1 -17171.726,E2 -17171.726} C_VEL
LIN {X 0,Y 284.628,Z 271.264,A -85,B 0,C 180,E1 -17171.982,E2 -17171.982} C_VEL
LIN {X 0,Y 294.174,Z 293.204,A -85,B 0,C 180,E1 -17173.382,E2 -17173.382} C_VEL
LIN {X 0,Y 295.456,Z 296.682,A -85,B 0,C 180,E1 -17173.573,E2 -17173.573} C_VEL
LIN {X 0,Y 294.31,Z 357.505,A -85,B 0,C 180,E1 -17175.082,E2 -17175.082} C_VEL
LIN {X 0,Y 293.878,Z 370.514,A -85,B 0,C 180,E1 -17175.679,E2 -17175.679} C_VEL
LIN {X 0,Y 293.292,Z 383.55,A -85,B 0,C 180,E1 -17176.578,E2 -17176.578} C_VEL
LIN {X 0,Y 292.318,Z 395.376,A -85,B 0,C 180,E1 -17177.681,E2 -17177.681} C_VEL
LIN {X 0,Y 291.078,Z 406.696,A -85,B 0,C 180,E1 -17179.04,E2 -17179.04} C_VEL
LIN {X 0,Y 289.944,Z 416.866,A -85,B 0,C 180,E1 -17180.584,E2 -17180.584} C_VEL
LIN {X 0,Y 288.737,Z 426.039,A -85,B 0,C 180,E1 -17182.307,E2 -17182.307} C_VEL
LIN {X 0,Y 287.427,Z 434.924,A -85,B 0,C 180,E1 -17184.388,E2 -17184.388} C_VEL
LIN {X 0,Y 286.3,Z 442.1,A -85,B 0,C 180,E1 -17186.482,E2 -17186.482} C_VEL
LIN {X 0,Y 285.453,Z 447.846,A -85,B 0,C 180,E1 -17188.59,E2 -17188.59} C_VEL
LIN {X 0,Y 284.826,Z 452.379,A -85,B 0,C 180,E1 -17190.707,E2 -17190.707} C_VEL
LIN {X 0,Y 284.261,Z 455.861,A -85,B 0,C 180,E1 -17192.835,E2 -17192.835} C_VEL
LIN {X 0,Y 284.149,Z 457.601,A -85,B 0,C 180,E1 -17194.256,E2 -17194.256} C_VEL
LIN {X 0,Y 284.132,Z 458.926,A -85,B 0,C 180,E1 -17195.679,E2 -17195.679} C_VEL
LIN {X 0,Y 284.136,Z 460.455,A -85,B 0,C 180,E1 -17198.535,E2 -17198.535} C_VEL
LIN {X 0,Y 284.263,Z 460.602,A -85,B 0,C 180,E1 -17199.966,E2 -17199.966} C_VEL
LIN {X 0,Y 284.741,Z 459.746,A -85,B 0,C 180,E1 -17202.835,E2 -17202.835} C_VEL
LIN {X 0,Y 285.145,Z 458.731,A -85,B 0,C 180,E1 -17204.269,E2 -17204.269} C_VEL
LIN {X 0,Y 286.131,Z 456.021,A -85,B 0,C 180,E1 -17206.677,E2 -17206.677} C_VEL
LIN {X 0,Y 287.44,Z 451.669,A -85,B 0,C 180,E1 -17209.274,E2 -17209.274} C_VEL
LIN {X 0,Y 288.796,Z 446.823,A -85,B 0,C 180,E1 -17211.41,E2 -17211.41} C_VEL
LIN {X 0,Y 290.447,Z 440.885,A -85,B 0,C 180,E1 -17213.456,E2 -17213.456} C_VEL
LIN {X 0,Y 292.068,Z 434.319,A -85,B 0,C 180,E1 -17215.285,E2 -17215.285} C_VEL
LIN {X 0,Y 294.141,Z 425.388,A -85,B 0,C 180,E1 -17217.275,E2 -17217.275} C_VEL
LIN {X 0,Y 296.107,Z 415.058,A -85,B 0,C 180,E1 -17219.115,E2 -17219.115} C_VEL
LIN {X 0,Y 297.814,Z 405.332,A -85,B 0,C 180,E1 -17220.489,E2 -17220.489} C_VEL
LIN {X 0,Y 299.277,Z 395.033,A -85,B 0,C 180,E1 -17221.662,E2 -17221.662} C_VEL
LIN {X 0,Y 300.646,Z 382.748,A -85,B 0,C 180,E1 -17222.741,E2 -17222.741} C_VEL
LIN {X 0,Y 301.464,Z 370.04,A -85,B 0,C 180,E1 -17223.58,E2 -17223.58} C_VEL
LIN {X 0,Y 301.973,Z 357.037,A -85,B 0,C 180,E1 -17224.14,E2 -17224.14} C_VEL
LIN {X 0,Y 303.031,Z 315.481,A -85,B 0,C 180,E1 -17225.173,E2 -17225.173} C_VEL
LIN {X 0,Y 303.259,Z 305.974,A -85,B 0,C 180,E1 -17225.406,E2 -17225.406} C_VEL
LIN {X 0,Y 293.912,Z 287.426,A -85,B 0,C 180,E1 -17227.057,E2 -17227.057} C_VEL
LIN {X 0,Y 285.984,Z 273.86,A -85,B 0,C 180,E1 -17228.504,E2 -17228.504} C_VEL
LIN {X 0,Y 284.437,Z 270.9,A -85,B 0,C 180,E1 -17228.857,E2 -17228.857} C_VEL
LIN {X 0,Y 284.304,Z 270.108,A -85,B 0,C 180,E1 -17229.196,E2 -17229.196} C_VEL
LIN {X 0,Y 284.236,Z 270.063,A -85,B 0,C 180,E1 -17232.116,E2 -17232.116} C_VEL
LIN {X 0,Y 284.236,Z 270.058,A -85,B 0,C 180,E1 -17236.185,E2 -17236.185} C_VEL
LIN {X 0,Y 284.283,Z 270.071,A -85,B 0,C 180,E1 -17240.029,E2 -17240.029} C_VEL
LIN {X 0,Y 284.317,Z 270.044,A -85,B 0,C 180,E1 -17243.611,E2 -17243.611} C_VEL
LIN {X 0,Y 284.305,Z 270.06,A -85,B 0,C 180,E1 -17247.19,E2 -17247.19} C_VEL
LIN {X 0,Y 284.311,Z 270.032,A -85,B 0,C 180,E1 -17250.37,E2 -17250.37} C_VEL
LIN {X 0,Y 284.303,Z 270.073,A -85,B 0,C 180,E1 -17253.579,E2 -17253.579} C_VEL
LIN {X 0,Y 284.307,Z 270.045,A -85,B 0,C 180,E1 -17255.902,E2 -17255.902} C_VEL
LIN {X 0,Y 283.67,Z 270.11,A -85,B 0,C 180,E1 -17257.086,E2 -17257.086} C_VEL
LIN {X 0,Y 280.814,Z 270.462,A -85,B 0,C 180,E1 -17259.013,E2 -17259.013} C_VEL
LIN {X 0,Y 278.4,Z 270.781,A -85,B 0,C 180,E1 -17260.578,E2 -17260.578} C_VEL
LIN {X 0,Y 277.406,Z 270.924,A -85,B 0,C 180,E1 -17261.792,E2 -17261.792} C_VEL
LIN {X 0,Y 277.349,Z 270.935,A -85,B 0,C 180,E1 -17262.203,E2 -17262.203} C_VEL
LIN {X 0,Y 277.426,Z 270.913,A -85,B 0,C 180,E1 -17265.325,E2 -17265.325} C_VEL
LIN {X 0,Y 277.454,Z 270.911,A -85,B 0,C 180,E1 -17269.786,E2 -17269.786} C_VEL
LIN {X 0,Y 277.595,Z 270.905,A -85,B 0,C 180,E1 -17272.727,E2 -17272.727} C_VEL
LIN {X 0,Y 277.806,Z 270.88,A -85,B 0,C 180,E1 -17278.55,E2 -17278.55} C_VEL
LIN {X 0,Y 277.801,Z 270.865,A -85,B 0,C 180,E1 -17281.449,E2 -17281.449} C_VEL
LIN {X 0,Y 277.594,Z 270.891,A -85,B 0,C 180,E1 -17287.272,E2 -17287.272} C_VEL
LIN {X 0,Y 277.451,Z 270.924,A -85,B 0,C 180,E1 -17290.213,E2 -17290.213} C_VEL
LIN {X 0,Y 277.405,Z 270.925,A -85,B 0,C 180,E1 -17294.675,E2 -17294.675} C_VEL
LIN {X 0,Y 277.325,Z 270.937,A -85,B 0,C 180,E1 -17299.235,E2 -17299.235} C_VEL
LIN {X 0,Y 277.278,Z 270.947,A -85,B 0,C 180,E1 -17303.925,E2 -17303.925} C_VEL
LIN {X 0,Y 277.234,Z 270.922,A -85,B 0,C 180,E1 -17307.47,E2 -17307.47} C_VEL
LIN {X 0,Y 277.225,Z 270.953,A -85,B 0,C 180,E1 -17310.466,E2 -17310.466} C_VEL
LIN {X 0,Y 277.243,Z 270.927,A -85,B 0,C 180,E1 -17313.896,E2 -17313.896} C_VEL
LIN {X 0,Y 277.248,Z 270.944,A -85,B 0,C 180,E1 -17317.472,E2 -17317.472} C_VEL
LIN {X 0,Y 277.181,Z 270.962,A -85,B 0,C 180,E1 -17321.242,E2 -17321.242} C_VEL
LIN {X 0,Y 277.171,Z 270.959,A -85,B 0,C 180,E1 -17325.233,E2 -17325.233} C_VEL
LIN {X 0,Y 277.208,Z 271.22,A -85,B 0,C 180,E1 -17327.459,E2 -17327.459} C_VEL
LIN {X 0,Y 280.404,Z 281.823,A -85,B 0,C 180,E1 -17330.985,E2 -17330.985} C_VEL
LIN {X 0,Y 283.223,Z 292.667,A -85,B 0,C 180,E1 -17334.281,E2 -17334.281} C_VEL
LIN {X 0,Y 285.456,Z 303.013,A -85,B 0,C 180,E1 -17337.204,E2 -17337.204} C_VEL
LIN {X 0,Y 286.017,Z 306.38,A -85,B 0,C 180,E1 -17338.11,E2 -17338.11} C_VEL
LIN {X 0,Y 285.772,Z 310.043,A -85,B 0,C 180,E1 -17338.905,E2 -17338.905} C_VEL
LIN {X 0,Y 290.862,Z 341.3,A -85,B 0,C 180,E1 -17340.499,E2 -17340.499} C_VEL
LIN {X 0,Y 293.969,Z 365.694,A -85,B 0,C 180,E1 -17341.563,E2 -17341.563} C_VEL
LIN {X 0,Y 295.056,Z 378.03,A -85,B 0,C 180,E1 -17342.031,E2 -17342.031} C_VEL
LIN {X 0,Y 293.46,Z 422.266,A -85,B 0,C 180,E1 -17343.126,E2 -17343.126} C_VEL
LIN {X 0,Y 292.389,Z 435.963,A -85,B 0,C 180,E1 -17343.742,E2 -17343.742} C_VEL
LIN {X 0,Y 290.711,Z 448.848,A -85,B 0,C 180,E1 -17344.589,E2 -17344.589} C_VEL
LIN {X 0,Y 288.394,Z 461.416,A -85,B 0,C 180,E1 -17345.718,E2 -17345.718} C_VEL
LIN {X 0,Y 286.072,Z 472.652,A -85,B 0,C 180,E1 -17347.045,E2 -17347.045} C_VEL
LIN {X 0,Y 283.861,Z 482.817,A -85,B 0,C 180,E1 -17348.581,E2 -17348.581} C_VEL
LIN {X 0,Y 281.653,Z 492.028,A -85,B 0,C 180,E1 -17350.314,E2 -17350.314} C_VEL
LIN {X 0,Y 279.557,Z 501.066,A -85,B 0,C 180,E1 -17352.441,E2 -17352.441} C_VEL
LIN {X 0,Y 278.279,Z 507.266,A -85,B 0,C 180,E1 -17354.247,E2 -17354.247} C_VEL
LIN {X 0,Y 276.818,Z 514.318,A -85,B 0,C 180,E1 -17356.791,E2 -17356.791} C_VEL
LIN {X 0,Y 276.046,Z 519.032,A -85,B 0,C 180,E1 -17358.992,E2 -17358.992} C_VEL
LIN {X 0,Y 275.787,Z 522.688,A -85,B 0,C 180,E1 -17361.205,E2 -17361.205} C_VEL
LIN {X 0,Y 275.911,Z 525.356,A -85,B 0,C 180,E1 -17363.418,E2 -17363.418} C_VEL
LIN {X 0,Y 276.147,Z 527.069,A -85,B 0,C 180,E1 -17365.621,E2 -17365.621} C_VEL
LIN {X 0,Y 276.419,Z 527.729,A -85,B 0,C 180,E1 -17367.085,E2 -17367.085} C_VEL
LIN {X 0,Y 276.476,Z 527.915,A -85,B 0,C 180,E1 -17368.543,E2 -17368.543} C_VEL
LIN {X 0,Y 276.601,Z 527.699,A -85,B 0,C 180,E1 -17369.999,E2 -17369.999} C_VEL
LIN {X 0,Y 276.53,Z 527.054,A -85,B 0,C 180,E1 -17371.456,E2 -17371.456} C_VEL
LIN {X 0,Y 276.535,Z 526.007,A -85,B 0,C 180,E1 -17372.913,E2 -17372.913} C_VEL
LIN {X 0,Y 276.194,Z 523.523,A -85,B 0,C 180,E1 -17375.109,E2 -17375.109} C_VEL
LIN {X 0,Y 276.003,Z 520.004,A -85,B 0,C 180,E1 -17377.314,E2 -17377.314} C_VEL
LIN {X 0,Y 276.004,Z 515.366,A -85,B 0,C 180,E1 -17379.526,E2 -17379.526} C_VEL
LIN {X 0,Y 276.435,Z 508.349,A -85,B 0,C 180,E1 -17382.107,E2 -17382.107} C_VEL
LIN {X 0,Y 277.18,Z 500.736,A -85,B 0,C 180,E1 -17384.312,E2 -17384.312} C_VEL
LIN {X 0,Y 278.348,Z 491.917,A -85,B 0,C 180,E1 -17386.37,E2 -17386.37} C_VEL
LIN {X 0,Y 279.595,Z 482.585,A -85,B 0,C 180,E1 -17388.122,E2 -17388.122} C_VEL
LIN {X 0,Y 280.973,Z 473.288,A -85,B 0,C 180,E1 -17389.544,E2 -17389.544} C_VEL
LIN {X 0,Y 282.675,Z 461.832,A -85,B 0,C 180,E1 -17390.939,E2 -17390.939} C_VEL
LIN {X 0,Y 284.116,Z 449.916,A -85,B 0,C 180,E1 -17392.065,E2 -17392.065} C_VEL
LIN {X 0,Y 285.316,Z 437.552,A -85,B 0,C 180,E1 -17392.922,E2 -17392.922} C_VEL
LIN {X 0,Y 286.162,Z 424.421,A -85,B 0,C 180,E1 -17393.542,E2 -17393.542} C_VEL
LIN {X 0,Y 286.842,Z 396.813,A -85,B 0,C 180,E1 -17394.275,E2 -17394.275} C_VEL
LIN {X 0,Y 287.266,Z 374.411,A -85,B 0,C 180,E1 -17394.83,E2 -17394.83} C_VEL
LIN {X 0,Y 282.998,Z 329.526,A -85,B 0,C 180,E1 -17396.353,E2 -17396.353} C_VEL
LIN {X 0,Y 280.968,Z 311.824,A -85,B 0,C 180,E1 -17397.034,E2 -17397.034} C_VEL
LIN {X 0,Y 282.734,Z 297.612,A -85,B 0,C 180,E1 -17400.221,E2 -17400.221} C_VEL
LIN {X 0,Y 281.661,Z 290.631,A -85,B 0,C 180,E1 -17401.965,E2 -17401.965} C_VEL
LIN {X 0,Y 278.845,Z 277.507,A -85,B 0,C 180,E1 -17405.427,E2 -17405.427} C_VEL
LIN {X 0,Y 277.298,Z 271.029,A -85,B 0,C 180,E1 -17407.275,E2 -17407.275} C_VEL
LIN {X 0,Y 277.178,Z 270.956,A -85,B 0,C 180,E1 -17411.24,E2 -17411.24} C_VEL
LIN {X 0,Y 277.167,Z 270.937,A -85,B 0,C 180,E1 -17415.231,E2 -17415.231} C_VEL
LIN {X 0,Y 277.177,Z 270.958,A -85,B 0,C 180,E1 -17418.758,E2 -17418.758} C_VEL
LIN {X 0,Y 277.246,Z 270.944,A -85,B 0,C 180,E1 -17422.527,E2 -17422.527} C_VEL
LIN {X 0,Y 277.238,Z 270.946,A -85,B 0,C 180,E1 -17426.103,E2 -17426.103} C_VEL
LIN {X 0,Y 277.22,Z 270.951,A -85,B 0,C 180,E1 -17429.534,E2 -17429.534} C_VEL
LIN {X 0,Y 277.281,Z 270.944,A -85,B 0,C 180,E1 -17432.856,E2 -17432.856} C_VEL
LIN {X 0,Y 277.273,Z 270.94,A -85,B 0,C 180,E1 -17436.075,E2 -17436.075} C_VEL
LIN {X 0,Y 277.275,Z 270.94,A -85,B 0,C 180,E1 -17440.761,E2 -17440.761} C_VEL
LIN {X 0,Y 277.399,Z 270.93,A -85,B 0,C 180,E1 -17445.324,E2 -17445.324} C_VEL
LIN {X 0,Y 277.447,Z 270.913,A -85,B 0,C 180,E1 -17449.787,E2 -17449.787} C_VEL
LIN {X 0,Y 277.588,Z 270.905,A -85,B 0,C 180,E1 -17452.728,E2 -17452.728} C_VEL
LIN {X 0,Y 277.794,Z 270.87,A -85,B 0,C 180,E1 -17458.551,E2 -17458.551} C_VEL
LIN {X 0,Y 277.798,Z 270.875,A -85,B 0,C 180,E1 -17461.45,E2 -17461.45} C_VEL
LIN {X 0,Y 277.581,Z 270.898,A -85,B 0,C 180,E1 -17467.273,E2 -17467.273} C_VEL
LIN {X 0,Y 277.443,Z 270.916,A -85,B 0,C 180,E1 -17470.214,E2 -17470.214} C_VEL
LIN {X 0,Y 277.4,Z 270.926,A -85,B 0,C 180,E1 -17474.676,E2 -17474.676} C_VEL
LIN {X 0,Y 277.276,Z 270.938,A -85,B 0,C 180,E1 -17479.239,E2 -17479.239} C_VEL
LIN {X 0,Y 277.252,Z 270.947,A -85,B 0,C 180,E1 -17483.928,E2 -17483.928} C_VEL
LIN {X 0,Y 277.228,Z 270.945,A -85,B 0,C 180,E1 -17487.47,E2 -17487.47} C_VEL
LIN {X 0,Y 277.222,Z 270.952,A -85,B 0,C 180,E1 -17490.467,E2 -17490.467} C_VEL
LIN {X 0,Y 277.24,Z 270.943,A -85,B 0,C 180,E1 -17493.897,E2 -17493.897} C_VEL
LIN {X 0,Y 277.245,Z 270.95,A -85,B 0,C 180,E1 -17497.474,E2 -17497.474} C_VEL
LIN {X 0,Y 277.178,Z 270.94,A -85,B 0,C 180,E1 -17501.243,E2 -17501.243} C_VEL
LIN {X 0,Y 277.169,Z 270.944,A -85,B 0,C 180,E1 -17505.234,E2 -17505.234} C_VEL
LIN {X 0,Y 277.18,Z 270.957,A -85,B 0,C 180,E1 -17508.76,E2 -17508.76} C_VEL
LIN {X 0,Y 277.247,Z 270.925,A -85,B 0,C 180,E1 -17512.529,E2 -17512.529} C_VEL
LIN {X 0,Y 277.244,Z 270.95,A -85,B 0,C 180,E1 -17516.105,E2 -17516.105} C_VEL
LIN {X 0,Y 277.227,Z 270.938,A -85,B 0,C 180,E1 -17519.536,E2 -17519.536} C_VEL
LIN {X 0,Y 277.249,Z 270.95,A -85,B 0,C 180,E1 -17522.854,E2 -17522.854} C_VEL
LIN {X 0,Y 277.26,Z 270.943,A -85,B 0,C 180,E1 -17526.074,E2 -17526.074} C_VEL
LIN {X 0,Y 277.269,Z 270.911,A -85,B 0,C 180,E1 -17530.762,E2 -17530.762} C_VEL
LIN {X 0,Y 277.363,Z 271.396,A -85,B 0,C 180,E1 -17531.227,E2 -17531.227} C_VEL
LIN {X 0,Y 277.922,Z 273.167,A -85,B 0,C 180,E1 -17531.446,E2 -17531.446} C_VEL
LIN {X 0,Y 285.827,Z 290.778,A -85,B 0,C 180,E1 -17532.631,E2 -17532.631} C_VEL
LIN {X 0,Y 288.857,Z 298.242,A -85,B 0,C 180,E1 -17533.082,E2 -17533.082} C_VEL
LIN {X 0,Y 287.699,Z 358.013,A -85,B 0,C 180,E1 -17534.595,E2 -17534.595} C_VEL
LIN {X 0,Y 287.243,Z 371.141,A -85,B 0,C 180,E1 -17535.205,E2 -17535.205} C_VEL
LIN {X 0,Y 286.649,Z 383.684,A -85,B 0,C 180,E1 -17536.08,E2 -17536.08} C_VEL
LIN {X 0,Y 285.649,Z 395.72,A -85,B 0,C 180,E1 -17537.208,E2 -17537.208} C_VEL
LIN {X 0,Y 284.355,Z 407.133,A -85,B 0,C 180,E1 -17538.597,E2 -17538.597} C_VEL
LIN {X 0,Y 283.162,Z 417.376,A -85,B 0,C 180,E1 -17540.176,E2 -17540.176} C_VEL
LIN {X 0,Y 282.055,Z 425.765,A -85,B 0,C 180,E1 -17541.763,E2 -17541.763} C_VEL
LIN {X 0,Y 280.858,Z 433.527,A -85,B 0,C 180,E1 -17543.535,E2 -17543.535} C_VEL
LIN {X 0,Y 279.577,Z 441.13,A -85,B 0,C 180,E1 -17545.676,E2 -17545.676} C_VEL
LIN {X 0,Y 278.657,Z 447.216,A -85,B 0,C 180,E1 -17547.833,E2 -17547.833} C_VEL
LIN {X 0,Y 277.94,Z 452.064,A -85,B 0,C 180,E1 -17550.001,E2 -17550.001} C_VEL
LIN {X 0,Y 277.362,Z 455.826,A -85,B 0,C 180,E1 -17552.179,E2 -17552.179} C_VEL
LIN {X 0,Y 277.102,Z 458.573,A -85,B 0,C 180,E1 -17554.364,E2 -17554.364} C_VEL
LIN {X 0,Y 277.077,Z 459.873,A -85,B 0,C 180,E1 -17555.824,E2 -17555.824} C_VEL
LIN {X 0,Y 277.1,Z 461.245,A -85,B 0,C 180,E1 -17558.446,E2 -17558.446} C_VEL
LIN {X 0,Y 277.237,Z 461.444,A -85,B 0,C 180,E1 -17560.222,E2 -17560.222} C_VEL
LIN {X 0,Y 277.796,Z 460.533,A -85,B 0,C 180,E1 -17563.162,E2 -17563.162} C_VEL
LIN {X 0,Y 278.223,Z 459.468,A -85,B 0,C 180,E1 -17564.632,E2 -17564.632} C_VEL
LIN {X 0,Y 279.229,Z 456.875,A -85,B 0,C 180,E1 -17566.972,E2 -17566.972} C_VEL
LIN {X 0,Y 280.702,Z 452.284,A -85,B 0,C 180,E1 -17569.755,E2 -17569.755} C_VEL
LIN {X 0,Y 282.128,Z 447.375,A -85,B 0,C 180,E1 -17571.942,E2 -17571.942} C_VEL
LIN {X 0,Y 283.95,Z 441.132,A -85,B 0,C 180,E1 -17574.104,E2 -17574.104} C_VEL
LIN {X 0,Y 285.957,Z 433.243,A -85,B 0,C 180,E1 -17576.256,E2 -17576.256} C_VEL
LIN {X 0,Y 288.01,Z 424.639,A -85,B 0,C 180,E1 -17578.128,E2 -17578.128} C_VEL
LIN {X 0,Y 289.862,Z 415.188,A -85,B 0,C 180,E1 -17579.804,E2 -17579.804} C_VEL
LIN {X 0,Y 291.608,Z 405.258,A -85,B 0,C 180,E1 -17581.209,E2 -17581.209} C_VEL
LIN {X 0,Y 293.11,Z 395.121,A -85,B 0,C 180,E1 -17582.359,E2 -17582.359} C_VEL
LIN {X 0,Y 294.471,Z 383.406,A -85,B 0,C 180,E1 -17583.396,E2 -17583.396} C_VEL
LIN {X 0,Y 295.276,Z 371.278,A -85,B 0,C 180,E1 -17584.215,E2 -17584.215} C_VEL
LIN {X 0,Y 295.858,Z 358.288,A -85,B 0,C 180,E1 -17584.794,E2 -17584.794} C_VEL
LIN {X 0,Y 296.808,Z 320.08,A -85,B 0,C 180,E1 -17585.774,E2 -17585.774} C_VEL
LIN {X 0,Y 297.203,Z 308.261,A -85,B 0,C 180,E1 -17586.058,E2 -17586.058} C_VEL
LIN {X 0,Y 288.416,Z 290.902,A -85,B 0,C 180,E1 -17587.669,E2 -17587.669} C_VEL
LIN {X 0,Y 280.283,Z 277.019,A -85,B 0,C 180,E1 -17589.212,E2 -17589.212} C_VEL
LIN {X 0,Y 277.444,Z 271.956,A -85,B 0,C 180,E1 -17589.82,E2 -17589.82} C_VEL
LIN {X 0,Y 277.255,Z 271.096,A -85,B 0,C 180,E1 -17590.104,E2 -17590.104} C_VEL
LIN {X 0,Y 277.191,Z 270.947,A -85,B 0,C 180,E1 -17593.201,E2 -17593.201} C_VEL
LIN {X 0,Y 277.191,Z 270.934,A -85,B 0,C 180,E1 -17597.33,E2 -17597.33} C_VEL
LIN {X 0,Y 277.249,Z 270.921,A -85,B 0,C 180,E1 -17601.796,E2 -17601.796} C_VEL
LIN {X 0,Y 277.276,Z 270.932,A -85,B 0,C 180,E1 -17604.34,E2 -17604.34} C_VEL
LIN {X 0,Y 277.236,Z 270.927,A -85,B 0,C 180,E1 -17607.835,E2 -17607.835} C_VEL
LIN {X 0,Y 277.265,Z 270.942,A -85,B 0,C 180,E1 -17612.518,E2 -17612.518} C_VEL
LIN {X 0,Y 277.28,Z 270.916,A -85,B 0,C 180,E1 -17616.075,E2 -17616.075} C_VEL
LIN {X 0,Y 277.34,Z 270.916,A -85,B 0,C 180,E1 -17620.765,E2 -17620.765} C_VEL
LIN {X 0,Y 277.349,Z 270.935,A -85,B 0,C 180,E1 -17622.203,E2 -17622.203} C_VEL
LIN {X 0,Y 276.747,Z 271.028,A -85,B 0,C 180,E1 -17623.416,E2 -17623.416} C_VEL
LIN {X 0,Y 273.925,Z 271.385,A -85,B 0,C 180,E1 -17625.392,E2 -17625.392} C_VEL
LIN {X 0,Y 271.496,Z 271.676,A -85,B 0,C 180,E1 -17626.998,E2 -17626.998} C_VEL
LIN {X 0,Y 270.456,Z 271.796,A -85,B 0,C 180,E1 -17628.243,E2 -17628.243} C_VEL
LIN {X 0,Y 270.375,Z 271.799,A -85,B 0,C 180,E1 -17628.665,E2 -17628.665} C_VEL
LIN {X 0,Y 270.557,Z 271.781,A -85,B 0,C 180,E1 -17632.537,E2 -17632.537} C_VEL
LIN {X 0,Y 270.77,Z 271.756,A -85,B 0,C 180,E1 -17638.512,E2 -17638.512} C_VEL
LIN {X 0,Y 270.766,Z 271.741,A -85,B 0,C 180,E1 -17641.487,E2 -17641.487} C_VEL
LIN {X 0,Y 270.556,Z 271.766,A -85,B 0,C 180,E1 -17647.462,E2 -17647.462} C_VEL
LIN {X 0,Y 270.403,Z 271.802,A -85,B 0,C 180,E1 -17650.482,E2 -17650.482} C_VEL
LIN {X 0,Y 270.374,Z 271.803,A -85,B 0,C 180,E1 -17655.066,E2 -17655.066} C_VEL
LIN {X 0,Y 270.276,Z 271.82,A -85,B 0,C 180,E1 -17659.757,E2 -17659.757} C_VEL
LIN {X 0,Y 270.221,Z 271.827,A -85,B 0,C 180,E1 -17664.591,E2 -17664.591} C_VEL
LIN {X 0,Y 270.182,Z 271.8,A -85,B 0,C 180,E1 -17667.919,E2 -17667.919} C_VEL
LIN {X 0,Y 270.166,Z 271.831,A -85,B 0,C 180,E1 -17671.35,E2 -17671.35} C_VEL
LIN {X 0,Y 270.195,Z 271.811,A -85,B 0,C 180,E1 -17674.906,E2 -17674.906} C_VEL
LIN {X 0,Y 270.196,Z 271.812,A -85,B 0,C 180,E1 -17678.711,E2 -17678.711} C_VEL
LIN {X 0,Y 270.145,Z 271.822,A -85,B 0,C 180,E1 -17683.245,E2 -17683.245} C_VEL
LIN {X 0,Y 270.165,Z 272.049,A -85,B 0,C 180,E1 -17686.513,E2 -17686.513} C_VEL
LIN {X 0,Y 273.58,Z 283.322,A -85,B 0,C 180,E1 -17690.414,E2 -17690.414} C_VEL
LIN {X 0,Y 276.452,Z 294.363,A -85,B 0,C 180,E1 -17693.881,E2 -17693.881} C_VEL
LIN {X 0,Y 278.577,Z 304.297,A -85,B 0,C 180,E1 -17696.77,E2 -17696.77} C_VEL
LIN {X 0,Y 279.308,Z 308.872,A -85,B 0,C 180,E1 -17697.972,E2 -17697.972} C_VEL
LIN {X 0,Y 281.601,Z 321.83,A -85,B 0,C 180,E1 -17698.728,E2 -17698.728} C_VEL
LIN {X 0,Y 285.663,Z 348.318,A -85,B 0,C 180,E1 -17700.051,E2 -17700.051} C_VEL
LIN {X 0,Y 288.574,Z 373.526,A -85,B 0,C 180,E1 -17701.144,E2 -17701.144} C_VEL
LIN {X 0,Y 288.887,Z 380.43,A -85,B 0,C 180,E1 -17701.38,E2 -17701.38} C_VEL
LIN {X 0,Y 287.348,Z 421.228,A -85,B 0,C 180,E1 -17702.408,E2 -17702.408} C_VEL
LIN {X 0,Y 286.23,Z 434.982,A -85,B 0,C 180,E1 -17703.033,E2 -17703.033} C_VEL
LIN {X 0,Y 284.511,Z 447.906,A -85,B 0,C 180,E1 -17703.896,E2 -17703.896} C_VEL
LIN {X 0,Y 282.284,Z 459.697,A -85,B 0,C 180,E1 -17704.96,E2 -17704.96} C_VEL
LIN {X 0,Y 279.824,Z 471.087,A -85,B 0,C 180,E1 -17706.306,E2 -17706.306} C_VEL
LIN {X 0,Y 277.502,Z 481.406,A -85,B 0,C 180,E1 -17707.869,E2 -17707.869} C_VEL
LIN {X 0,Y 274.966,Z 491.54,A -85,B 0,C 180,E1 -17709.815,E2 -17709.815} C_VEL
LIN {X 0,Y 272.759,Z 500.514,A -85,B 0,C 180,E1 -17711.989,E2 -17711.989} C_VEL
LIN {X 0,Y 271.16,Z 507.788,A -85,B 0,C 180,E1 -17714.208,E2 -17714.208} C_VEL
LIN {X 0,Y 269.855,Z 513.637,A -85,B 0,C 180,E1 -17716.444,E2 -17716.444} C_VEL
LIN {X 0,Y 269.014,Z 518.307,A -85,B 0,C 180,E1 -17718.7,E2 -17718.7} C_VEL
LIN {X 0,Y 268.71,Z 521.93,A -85,B 0,C 180,E1 -17720.971,E2 -17720.971} C_VEL
LIN {X 0,Y 268.846,Z 524.719,A -85,B 0,C 180,E1 -17723.399,E2 -17723.399} C_VEL
LIN {X 0,Y 269.057,Z 526.256,A -85,B 0,C 180,E1 -17725.505,E2 -17725.505} C_VEL
LIN {X 0,Y 269.333,Z 526.89,A -85,B 0,C 180,E1 -17727.008,E2 -17727.008} C_VEL
LIN {X 0,Y 269.428,Z 527.057,A -85,B 0,C 180,E1 -17728.505,E2 -17728.505} C_VEL
LIN {X 0,Y 269.552,Z 526.823,A -85,B 0,C 180,E1 -17729.999,E2 -17729.999} C_VEL
LIN {X 0,Y 269.482,Z 526.161,A -85,B 0,C 180,E1 -17731.494,E2 -17731.494} C_VEL
LIN {X 0,Y 269.484,Z 525.087,A -85,B 0,C 180,E1 -17732.989,E2 -17732.989} C_VEL
LIN {X 0,Y 269.11,Z 522.567,A -85,B 0,C 180,E1 -17735.244,E2 -17735.244} C_VEL
LIN {X 0,Y 268.921,Z 519.007,A -85,B 0,C 180,E1 -17737.508,E2 -17737.508} C_VEL
LIN {X 0,Y 268.944,Z 514.323,A -85,B 0,C 180,E1 -17739.779,E2 -17739.779} C_VEL
LIN {X 0,Y 269.437,Z 507.239,A -85,B 0,C 180,E1 -17742.426,E2 -17742.426} C_VEL
LIN {X 0,Y 270.253,Z 499.573,A -85,B 0,C 180,E1 -17744.687,E2 -17744.687} C_VEL
LIN {X 0,Y 271.384,Z 491.449,A -85,B 0,C 180,E1 -17746.628,E2 -17746.628} C_VEL
LIN {X 0,Y 272.867,Z 481.255,A -85,B 0,C 180,E1 -17748.585,E2 -17748.585} C_VEL
LIN {X 0,Y 274.476,Z 470.543,A -85,B 0,C 180,E1 -17750.222,E2 -17750.222} C_VEL
LIN {X 0,Y 276.217,Z 458.608,A -85,B 0,C 180,E1 -17751.649,E2 -17751.649} C_VEL
LIN {X 0,Y 277.69,Z 446.961,A -85,B 0,C 180,E1 -17752.702,E2 -17752.702} C_VEL
LIN {X 0,Y 278.818,Z 433.743,A -85,B 0,C 180,E1 -17753.586,E2 -17753.586} C_VEL
LIN {X 0,Y 279.641,Z 420.469,A -85,B 0,C 180,E1 -17754.159,E2 -17754.159} C_VEL
LIN {X 0,Y 280.643,Z 375.297,A -85,B 0,C 180,E1 -17755.318,E2 -17755.318} C_VEL
LIN {X 0,Y 276.575,Z 331.334,A -85,B 0,C 180,E1 -17756.846,E2 -17756.846} C_VEL
LIN {X 0,Y 274.225,Z 311.124,A -85,B 0,C 180,E1 -17757.639,E2 -17757.639} C_VEL
LIN {X 0,Y 275.07,Z 304.777,A -85,B 0,C 180,E1 -17759.04,E2 -17759.04} C_VEL
LIN {X 0,Y 275.782,Z 297.989,A -85,B 0,C 180,E1 -17760.641,E2 -17760.641} C_VEL
LIN {X 0,Y 273.76,Z 287.078,A -85,B 0,C 180,E1 -17763.499,E2 -17763.499} C_VEL
LIN {X 0,Y 270.95,Z 274.695,A -85,B 0,C 180,E1 -17766.926,E2 -17766.926} C_VEL
LIN {X 0,Y 270.243,Z 271.909,A -85,B 0,C 180,E1 -17767.788,E2 -17767.788} C_VEL
LIN {X 0,Y 270.145,Z 271.834,A -85,B 0,C 180,E1 -17772.561,E2 -17772.561} C_VEL
LIN {X 0,Y 270.141,Z 271.822,A -85,B 0,C 180,E1 -17776.754,E2 -17776.754} C_VEL
LIN {X 0,Y 270.201,Z 271.82,A -85,B 0,C 180,E1 -17781.373,E2 -17781.373} C_VEL
LIN {X 0,Y 270.19,Z 271.829,A -85,B 0,C 180,E1 -17785.093,E2 -17785.093} C_VEL
LIN {X 0,Y 270.163,Z 271.826,A -85,B 0,C 180,E1 -17789.141,E2 -17789.141} C_VEL
LIN {X 0,Y 270.189,Z 271.827,A -85,B 0,C 180,E1 -17792.172,E2 -17792.172} C_VEL
LIN {X 0,Y 270.219,Z 271.819,A -85,B 0,C 180,E1 -17795.542,E2 -17795.542} C_VEL
LIN {X 0,Y 270.214,Z 271.823,A -85,B 0,C 180,E1 -17800.238,E2 -17800.238} C_VEL
LIN {X 0,Y 270.359,Z 271.809,A -85,B 0,C 180,E1 -17804.933,E2 -17804.933} C_VEL
LIN {X 0,Y 270.4,Z 271.79,A -85,B 0,C 180,E1 -17809.518,E2 -17809.518} C_VEL
LIN {X 0,Y 270.55,Z 271.779,A -85,B 0,C 180,E1 -17812.537,E2 -17812.537} C_VEL
LIN {X 0,Y 270.76,Z 271.745,A -85,B 0,C 180,E1 -17818.513,E2 -17818.513} C_VEL
LIN {X 0,Y 270.762,Z 271.751,A -85,B 0,C 180,E1 -17821.488,E2 -17821.488} C_VEL
LIN {X 0,Y 270.542,Z 271.774,A -85,B 0,C 180,E1 -17827.463,E2 -17827.463} C_VEL
LIN {X 0,Y 270.378,Z 271.798,A -85,B 0,C 180,E1 -17830.484,E2 -17830.484} C_VEL
LIN {X 0,Y 270.359,Z 271.802,A -85,B 0,C 180,E1 -17835.068,E2 -17835.068} C_VEL
LIN {X 0,Y 270.215,Z 271.819,A -85,B 0,C 180,E1 -17839.763,E2 -17839.763} C_VEL
LIN {X 0,Y 270.177,Z 271.822,A -85,B 0,C 180,E1 -17844.438,E2 -17844.438} C_VEL
LIN {X 0,Y 270.177,Z 271.825,A -85,B 0,C 180,E1 -17847.92,E2 -17847.92} C_VEL
LIN {X 0,Y 270.162,Z 271.83,A -85,B 0,C 180,E1 -17851.352,E2 -17851.352} C_VEL
LIN {X 0,Y 270.191,Z 271.823,A -85,B 0,C 180,E1 -17854.908,E2 -17854.908} C_VEL
LIN {X 0,Y 270.193,Z 271.824,A -85,B 0,C 180,E1 -17858.712,E2 -17858.712} C_VEL
LIN {X 0,Y 270.142,Z 271.8,A -85,B 0,C 180,E1 -17863.246,E2 -17863.246} C_VEL
LIN {X 0,Y 270.147,Z 271.832,A -85,B 0,C 180,E1 -17867.439,E2 -17867.439} C_VEL
LIN {X 0,Y 270.19,Z 271.812,A -85,B 0,C 180,E1 -17871.373,E2 -17871.373} C_VEL
LIN {X 0,Y 270.195,Z 271.822,A -85,B 0,C 180,E1 -17875.095,E2 -17875.095} C_VEL
LIN {X 0,Y 270.17,Z 271.818,A -85,B 0,C 180,E1 -17879.143,E2 -17879.143} C_VEL
LIN {X 0,Y 270.187,Z 271.83,A -85,B 0,C 180,E1 -17882.179,E2 -17882.179} C_VEL
LIN {X 0,Y 270.184,Z 271.819,A -85,B 0,C 180,E1 -17885.564,E2 -17885.564} C_VEL
LIN {X 0,Y 270.244,Z 271.903,A -85,B 0,C 180,E1 -17890.359,E2 -17890.359} C_VEL
LIN {X 0,Y 270.413,Z 272.709,A -85,B 0,C 180,E1 -17890.665,E2 -17890.665} C_VEL
LIN {X 0,Y 274.807,Z 282.301,A -85,B 0,C 180,E1 -17891.415,E2 -17891.415} C_VEL
LIN {X 0,Y 282.333,Z 300.004,A -85,B 0,C 180,E1 -17892.579,E2 -17892.579} C_VEL
LIN {X 0,Y 281.096,Z 357.082,A -85,B 0,C 180,E1 -17894.038,E2 -17894.038} C_VEL
LIN {X 0,Y 280.712,Z 369.496,A -85,B 0,C 180,E1 -17894.574,E2 -17894.574} C_VEL
LIN {X 0,Y 280.217,Z 381.581,A -85,B 0,C 180,E1 -17895.383,E2 -17895.383} C_VEL
LIN {X 0,Y 279.149,Z 394.342,A -85,B 0,C 180,E1 -17896.534,E2 -17896.534} C_VEL
LIN {X 0,Y 277.942,Z 404.967,A -85,B 0,C 180,E1 -17897.775,E2 -17897.775} C_VEL
LIN {X 0,Y 276.645,Z 415.784,A -85,B 0,C 180,E1 -17899.387,E2 -17899.387} C_VEL
LIN {X 0,Y 275.376,Z 425.446,A -85,B 0,C 180,E1 -17901.193,E2 -17901.193} C_VEL
LIN {X 0,Y 274.107,Z 433.402,A -85,B 0,C 180,E1 -17903.005,E2 -17903.005} C_VEL
LIN {X 0,Y 272.753,Z 441.231,A -85,B 0,C 180,E1 -17905.197,E2 -17905.197} C_VEL
LIN {X 0,Y 271.979,Z 446.502,A -85,B 0,C 180,E1 -17907.038,E2 -17907.038} C_VEL
LIN {X 0,Y 271.136,Z 451.692,A -85,B 0,C 180,E1 -17909.258,E2 -17909.258} C_VEL
LIN {X 0,Y 270.512,Z 455.742,A -85,B 0,C 180,E1 -17911.489,E2 -17911.489} C_VEL
LIN {X 0,Y 270.141,Z 457.88,A -85,B 0,C 180,E1 -17912.983,E2 -17912.983} C_VEL
LIN {X 0,Y 270.055,Z 459.542,A -85,B 0,C 180,E1 -17914.478,E2 -17914.478} C_VEL
LIN {X 0,Y 270.026,Z 460.818,A -85,B 0,C 180,E1 -17915.976,E2 -17915.976} C_VEL
LIN {X 0,Y 270.061,Z 462.095,A -85,B 0,C 180,E1 -17918.539,E2 -17918.539} C_VEL
LIN {X 0,Y 270.231,Z 462.286,A -85,B 0,C 180,E1 -17920.49,E2 -17920.49} C_VEL
LIN {X 0,Y 270.865,Z 461.318,A -85,B 0,C 180,E1 -17923.505,E2 -17923.505} C_VEL
LIN {X 0,Y 271.314,Z 460.203,A -85,B 0,C 180,E1 -17925.013,E2 -17925.013} C_VEL
LIN {X 0,Y 272.347,Z 457.718,A -85,B 0,C 180,E1 -17927.291,E2 -17927.291} C_VEL
LIN {X 0,Y 273.504,Z 454.299,A -85,B 0,C 180,E1 -17929.515,E2 -17929.515} C_VEL
LIN {X 0,Y 274.943,Z 449.712,A -85,B 0,C 180,E1 -17931.755,E2 -17931.755} C_VEL
LIN {X 0,Y 277.086,Z 442.731,A -85,B 0,C 180,E1 -17934.341,E2 -17934.341} C_VEL
LIN {X 0,Y 279.144,Z 435.079,A -85,B 0,C 180,E1 -17936.544,E2 -17936.544} C_VEL
LIN {X 0,Y 281.55,Z 425.493,A -85,B 0,C 180,E1 -17938.696,E2 -17938.696} C_VEL
LIN {X 0,Y 283.433,Z 416.391,A -85,B 0,C 180,E1 -17940.346,E2 -17940.346} C_VEL
LIN {X 0,Y 285.44,Z 405.142,A -85,B 0,C 180,E1 -17941.962,E2 -17941.962} C_VEL
LIN {X 0,Y 287.184,Z 393.83,A -85,B 0,C 180,E1 -17943.222,E2 -17943.222} C_VEL
LIN {X 0,Y 288.487,Z 382.714,A -85,B 0,C 180,E1 -17944.183,E2 -17944.183} C_VEL
LIN {X 0,Y 289.311,Z 369.87,A -85,B 0,C 180,E1 -17945.023,E2 -17945.023} C_VEL
LIN {X 0,Y 289.775,Z 357.563,A -85,B 0,C 180,E1 -17945.543,E2 -17945.543} C_VEL
LIN {X 0,Y 290.966,Z 316.006,A -85,B 0,C 180,E1 -17946.607,E2 -17946.607} C_VEL
LIN {X 0,Y 291.083,Z 310.295,A -85,B 0,C 180,E1 -17946.757,E2 -17946.757} C_VEL
LIN {X 0,Y 282.928,Z 294.238,A -85,B 0,C 180,E1 -17948.312,E2 -17948.312} C_VEL
LIN {X 0,Y 274.062,Z 279.094,A -85,B 0,C 180,E1 -17950.074,E2 -17950.074} C_VEL
LIN {X 0,Y 271.913,Z 275.694,A -85,B 0,C 180,E1 -17950.517,E2 -17950.517} C_VEL
LIN {X 0,Y 270.388,Z 272.948,A -85,B 0,C 180,E1 -17950.874,E2 -17950.874} C_VEL
LIN {X 0,Y 270.172,Z 271.951,A -85,B 0,C 180,E1 -17951.202,E2 -17951.202} C_VEL
LIN {X 0,Y 270.128,Z 271.823,A -85,B 0,C 180,E1 -17955.374,E2 -17955.374} C_VEL
LIN {X 0,Y 270.148,Z 271.835,A -85,B 0,C 180,E1 -17959.429,E2 -17959.429} C_VEL
LIN {X 0,Y 270.206,Z 271.797,A -85,B 0,C 180,E1 -17963.256,E2 -17963.256} C_VEL
LIN {X 0,Y 270.2,Z 271.822,A -85,B 0,C 180,E1 -17966.891,E2 -17966.891} C_VEL
LIN {X 0,Y 270.158,Z 271.793,A -85,B 0,C 180,E1 -17970.378,E2 -17970.378} C_VEL
LIN {X 0,Y 270.199,Z 271.831,A -85,B 0,C 180,E1 -17973.757,E2 -17973.757} C_VEL
LIN {X 0,Y 270.198,Z 271.781,A -85,B 0,C 180,E1 -17977.035,E2 -17977.035} C_VEL
LIN {X 0,Y 270.287,Z 271.784,A -85,B 0,C 180,E1 -17980.243,E2 -17980.243} C_VEL
LIN {X 0,Y 270.394,Z 271.79,A -85,B 0,C 180,E1 -17984.934,E2 -17984.934} C_VEL
LIN {X 0,Y 270.375,Z 271.799,A -85,B 0,C 180,E1 -17988.665,E2 -17988.665} C_VEL
LIN {X 0,Y 269.724,Z 271.875,A -85,B 0,C 180,E1 -17989.909,E2 -17989.909} C_VEL
LIN {X 0,Y 266.904,Z 272.227,A -85,B 0,C 180,E1 -17991.939,E2 -17991.939} C_VEL
LIN {X 0,Y 264.489,Z 272.54,A -85,B 0,C 180,E1 -17993.588,E2 -17993.588} C_VEL
LIN {X 0,Y 263.433,Z 272.662,A -85,B 0,C 180,E1 -17994.866,E2 -17994.866} C_VEL
LIN {X 0,Y 263.337,Z 272.669,A -85,B 0,C 180,E1 -17995.299,E2 -17995.299} C_VEL
LIN {X 0,Y 263.733,Z 272.633,A -85,B 0,C 180,E1 -17998.473,E2 -17998.473} C_VEL
LIN {X 0,Y 263.73,Z 272.617,A -85,B 0,C 180,E1 -18001.527,E2 -18001.527} C_VEL
LIN {X 0,Y 263.521,Z 272.642,A -85,B 0,C 180,E1 -18007.663,E2 -18007.663} C_VEL
LIN {X 0,Y 263.342,Z 272.682,A -85,B 0,C 180,E1 -18010.767,E2 -18010.767} C_VEL
LIN {X 0,Y 263.32,Z 272.685,A -85,B 0,C 180,E1 -18015.48,E2 -18015.48} C_VEL
LIN {X 0,Y 263.24,Z 272.695,A -85,B 0,C 180,E1 -18020.308,E2 -18020.308} C_VEL
LIN {X 0,Y 263.158,Z 272.697,A -85,B 0,C 180,E1 -18025.296,E2 -18025.296} C_VEL
LIN {X 0,Y 263.115,Z 272.686,A -85,B 0,C 180,E1 -18028.737,E2 -18028.737} C_VEL
LIN {X 0,Y 263.123,Z 272.696,A -85,B 0,C 180,E1 -18032.289,E2 -18032.289} C_VEL
LIN {X 0,Y 263.154,Z 272.705,A -85,B 0,C 180,E1 -18035.983,E2 -18035.983} C_VEL
LIN {X 0,Y 263.089,Z 272.702,A -85,B 0,C 180,E1 -18039.875,E2 -18039.875} C_VEL
LIN {X 0,Y 263.079,Z 272.706,A -85,B 0,C 180,E1 -18043.993,E2 -18043.993} C_VEL
LIN {X 0,Y 263.114,Z 272.913,A -85,B 0,C 180,E1 -18045.514,E2 -18045.514} C_VEL
LIN {X 0,Y 266.761,Z 284.854,A -85,B 0,C 180,E1 -18049.82,E2 -18049.82} C_VEL
LIN {X 0,Y 269.703,Z 296.101,A -85,B 0,C 180,E1 -18053.472,E2 -18053.472} C_VEL
LIN {X 0,Y 271.728,Z 305.488,A -85,B 0,C 180,E1 -18056.291,E2 -18056.291} C_VEL
LIN {X 0,Y 272.238,Z 307.988,A -85,B 0,C 180,E1 -18056.924,E2 -18056.924} C_VEL
LIN {X 0,Y 273.91,Z 312.836,A -85,B 0,C 180,E1 -18057.361,E2 -18057.361} C_VEL
LIN {X 0,Y 278.359,Z 339.908,A -85,B 0,C 180,E1 -18058.834,E2 -18058.834} C_VEL
LIN {X 0,Y 281.843,Z 367.307,A -85,B 0,C 180,E1 -18060.122,E2 -18060.122} C_VEL
LIN {X 0,Y 282.846,Z 380.204,A -85,B 0,C 180,E1 -18060.631,E2 -18060.631} C_VEL
LIN {X 0,Y 281.295,Z 420.192,A -85,B 0,C 180,E1 -18061.66,E2 -18061.66} C_VEL
LIN {X 0,Y 280.089,Z 434.003,A -85,B 0,C 180,E1 -18062.291,E2 -18062.291} C_VEL
LIN {X 0,Y 278.487,Z 445.893,A -85,B 0,C 180,E1 -18063.084,E2 -18063.084} C_VEL
LIN {X 0,Y 276.217,Z 457.978,A -85,B 0,C 180,E1 -18064.169,E2 -18064.169} C_VEL
LIN {X 0,Y 273.706,Z 469.525,A -85,B 0,C 180,E1 -18065.541,E2 -18065.541} C_VEL
LIN {X 0,Y 271.175,Z 479.965,A -85,B 0,C 180,E1 -18067.123,E2 -18067.123} C_VEL
LIN {X 0,Y 268.728,Z 489.404,A -85,B 0,C 180,E1 -18068.924,E2 -18068.924} C_VEL
LIN {X 0,Y 266.292,Z 498.58,A -85,B 0,C 180,E1 -18071.137,E2 -18071.137} C_VEL
LIN {X 0,Y 264.513,Z 505.474,A -85,B 0,C 180,E1 -18073.209,E2 -18073.209} C_VEL
LIN {X 0,Y 263.257,Z 511.143,A -85,B 0,C 180,E1 -18075.308,E2 -18075.308} C_VEL
LIN {X 0,Y 262.229,Z 516.151,A -85,B 0,C 180,E1 -18077.619,E2 -18077.619} C_VEL
LIN {X 0,Y 261.699,Z 520.068,A -85,B 0,C 180,E1 -18079.947,E2 -18079.947} C_VEL
LIN {X 0,Y 261.664,Z 522.997,A -85,B 0,C 180,E1 -18082.282,E2 -18082.282} C_VEL
LIN {X 0,Y 261.825,Z 524.424,A -85,B 0,C 180,E1 -18083.836,E2 -18083.836} C_VEL
LIN {X 0,Y 261.97,Z 525.443,A -85,B 0,C 180,E1 -18085.383,E2 -18085.383} C_VEL
LIN {X 0,Y 262.25,Z 526.045,A -85,B 0,C 180,E1 -18086.927,E2 -18086.927} C_VEL
LIN {X 0,Y 262.379,Z 526.198,A -85,B 0,C 180,E1 -18088.465,E2 -18088.465} C_VEL
LIN {X 0,Y 262.503,Z 525.948,A -85,B 0,C 180,E1 -18089.999,E2 -18089.999} C_VEL
LIN {X 0,Y 262.434,Z 525.267,A -85,B 0,C 180,E1 -18091.534,E2 -18091.534} C_VEL
LIN {X 0,Y 262.412,Z 524.158,A -85,B 0,C 180,E1 -18093.07,E2 -18093.07} C_VEL
LIN {X 0,Y 262.031,Z 521.605,A -85,B 0,C 180,E1 -18095.386,E2 -18095.386} C_VEL
LIN {X 0,Y 261.829,Z 518.002,A -85,B 0,C 180,E1 -18097.712,E2 -18097.712} C_VEL
LIN {X 0,Y 261.904,Z 513.272,A -85,B 0,C 180,E1 -18100.044,E2 -18100.044} C_VEL
LIN {X 0,Y 262.31,Z 507.27,A -85,B 0,C 180,E1 -18102.376,E2 -18102.376} C_VEL
LIN {X 0,Y 263.118,Z 499.787,A -85,B 0,C 180,E1 -18104.698,E2 -18104.698} C_VEL
LIN {X 0,Y 264.147,Z 492.321,A -85,B 0,C 180,E1 -18106.59,E2 -18106.59} C_VEL
LIN {X 0,Y 265.527,Z 483.032,A -85,B 0,C 180,E1 -18108.518,E2 -18108.518} C_VEL
LIN {X 0,Y 267.002,Z 474.187,A -85,B 0,C 180,E1 -18110.009,E2 -18110.009} C_VEL
LIN {X 0,Y 268.653,Z 463.424,A -85,B 0,C 180,E1 -18111.483,E2 -18111.483} C_VEL
LIN {X 0,Y 270.293,Z 451.39,A -85,B 0,C 180,E1 -18112.752,E2 -18112.752} C_VEL
LIN {X 0,Y 271.691,Z 438.865,A -85,B 0,C 180,E1 -18113.737,E2 -18113.737} C_VEL
LIN {X 0,Y 272.68,Z 425.842,A -85,B 0,C 180,E1 -18114.456,E2 -18114.456} C_VEL
LIN {X 0,Y 273.227,Z 411.63,A -85,B 0,C 180,E1 -18114.918,E2 -18114.918} C_VEL
LIN {X 0,Y 273.973,Z 375.484,A -85,B 0,C 180,E1 -18115.853,E2 -18115.853} C_VEL
LIN {X 0,Y 270.053,Z 332.248,A -85,B 0,C 180,E1 -18117.398,E2 -18117.398} C_VEL
LIN {X 0,Y 267.523,Z 310.157,A -85,B 0,C 180,E1 -18118.3,E2 -18118.3} C_VEL
LIN {X 0,Y 268.873,Z 299.426,A -85,B 0,C 180,E1 -18120.813,E2 -18120.813} C_VEL
LIN {X 0,Y 266.998,Z 289.229,A -85,B 0,C 180,E1 -18123.555,E2 -18123.555} C_VEL
LIN {X 0,Y 264.233,Z 276.85,A -85,B 0,C 180,E1 -18127.067,E2 -18127.067} C_VEL
LIN {X 0,Y 263.158,Z 272.769,A -85,B 0,C 180,E1 -18128.37,E2 -18128.37} C_VEL
LIN {X 0,Y 263.103,Z 272.713,A -85,B 0,C 180,E1 -18131.895,E2 -18131.895} C_VEL
LIN {X 0,Y 263.072,Z 272.695,A -85,B 0,C 180,E1 -18136.16,E2 -18136.16} C_VEL
LIN {X 0,Y 263.106,Z 272.706,A -85,B 0,C 180,E1 -18140.77,E2 -18140.77} C_VEL
LIN {X 0,Y 263.15,Z 272.705,A -85,B 0,C 180,E1 -18144.016,E2 -18144.016} C_VEL
LIN {X 0,Y 263.118,Z 272.696,A -85,B 0,C 180,E1 -18147.71,E2 -18147.71} C_VEL
LIN {X 0,Y 263.134,Z 272.706,A -85,B 0,C 180,E1 -18151.807,E2 -18151.807} C_VEL
LIN {X 0,Y 263.181,Z 272.693,A -85,B 0,C 180,E1 -18155.218,E2 -18155.218} C_VEL
LIN {X 0,Y 263.2,Z 272.696,A -85,B 0,C 180,E1 -18159.689,E2 -18159.689} C_VEL
LIN {X 0,Y 263.301,Z 272.683,A -85,B 0,C 180,E1 -18164.519,E2 -18164.519} C_VEL
LIN {X 0,Y 263.34,Z 272.67,A -85,B 0,C 180,E1 -18169.233,E2 -18169.233} C_VEL
LIN {X 0,Y 263.515,Z 272.653,A -85,B 0,C 180,E1 -18172.337,E2 -18172.337} C_VEL
LIN {X 0,Y 263.724,Z 272.62,A -85,B 0,C 180,E1 -18178.473,E2 -18178.473} C_VEL
LIN {X 0,Y 263.725,Z 272.628,A -85,B 0,C 180,E1 -18181.527,E2 -18181.527} C_VEL
LIN {X 0,Y 263.504,Z 272.65,A -85,B 0,C 180,E1 -18187.664,E2 -18187.664} C_VEL
LIN {X 0,Y 263.324,Z 272.68,A -85,B 0,C 180,E1 -18190.768,E2 -18190.768} C_VEL
LIN {X 0,Y 263.302,Z 272.681,A -85,B 0,C 180,E1 -18195.481,E2 -18195.481} C_VEL
LIN {X 0,Y 263.201,Z 272.697,A -85,B 0,C 180,E1 -18200.312,E2 -18200.312} C_VEL
LIN {X 0,Y 263.114,Z 272.7,A -85,B 0,C 180,E1 -18205.302,E2 -18205.302} C_VEL
LIN {X 0,Y 263.111,Z 272.709,A -85,B 0,C 180,E1 -18208.738,E2 -18208.738} C_VEL
LIN {X 0,Y 263.12,Z 272.702,A -85,B 0,C 180,E1 -18212.291,E2 -18212.291} C_VEL
LIN {X 0,Y 263.151,Z 272.706,A -85,B 0,C 180,E1 -18215.985,E2 -18215.985} C_VEL
LIN {X 0,Y 263.086,Z 272.702,A -85,B 0,C 180,E1 -18219.877,E2 -18219.877} C_VEL
LIN {X 0,Y 263.072,Z 272.682,A -85,B 0,C 180,E1 -18223.996,E2 -18223.996} C_VEL
LIN {X 0,Y 263.077,Z 272.714,A -85,B 0,C 180,E1 -18228.419,E2 -18228.419} C_VEL
LIN {X 0,Y 263.127,Z 272.683,A -85,B 0,C 180,E1 -18232.099,E2 -18232.099} C_VEL
LIN {X 0,Y 263.15,Z 272.706,A -85,B 0,C 180,E1 -18235.887,E2 -18235.887} C_VEL
LIN {X 0,Y 263.108,Z 272.694,A -85,B 0,C 180,E1 -18239.503,E2 -18239.503} C_VEL
LIN {X 0,Y 263.113,Z 272.712,A -85,B 0,C 180,E1 -18242.995,E2 -18242.995} C_VEL
LIN {X 0,Y 263.117,Z 272.706,A -85,B 0,C 180,E1 -18246.382,E2 -18246.382} C_VEL
LIN {X 0,Y 263.211,Z 272.789,A -85,B 0,C 180,E1 -18249.69,E2 -18249.69} C_VEL
LIN {X 0,Y 263.408,Z 273.763,A -85,B 0,C 180,E1 -18250.006,E2 -18250.006} C_VEL
LIN {X 0,Y 271.204,Z 290.822,A -85,B 0,C 180,E1 -18251.315,E2 -18251.315} C_VEL
LIN {X 0,Y 275.721,Z 301.53,A -85,B 0,C 180,E1 -18252.036,E2 -18252.036} C_VEL
LIN {X 0,Y 274.52,Z 359.067,A -85,B 0,C 180,E1 -18253.553,E2 -18253.553} C_VEL
LIN {X 0,Y 274.017,Z 372.393,A -85,B 0,C 180,E1 -18254.187,E2 -18254.187} C_VEL
LIN {X 0,Y 273.366,Z 385.042,A -85,B 0,C 180,E1 -18255.103,E2 -18255.103} C_VEL
LIN {X 0,Y 272.361,Z 396.358,A -85,B 0,C 180,E1 -18256.192,E2 -18256.192} C_VEL
LIN {X 0,Y 270.964,Z 407.995,A -85,B 0,C 180,E1 -18257.645,E2 -18257.645} C_VEL
LIN {X 0,Y 269.647,Z 418.382,A -85,B 0,C 180,E1 -18259.299,E2 -18259.299} C_VEL
LIN {X 0,Y 268.446,Z 426.882,A -85,B 0,C 180,E1 -18260.963,E2 -18260.963} C_VEL
LIN {X 0,Y 267.126,Z 434.743,A -85,B 0,C 180,E1 -18262.822,E2 -18262.822} C_VEL
LIN {X 0,Y 265.754,Z 442.461,A -85,B 0,C 180,E1 -18265.07,E2 -18265.07} C_VEL
LIN {X 0,Y 264.956,Z 447.682,A -85,B 0,C 180,E1 -18266.96,E2 -18266.96} C_VEL
LIN {X 0,Y 264.094,Z 452.804,A -85,B 0,C 180,E1 -18269.238,E2 -18269.238} C_VEL
LIN {X 0,Y 263.433,Z 456.799,A -85,B 0,C 180,E1 -18271.529,E2 -18271.529} C_VEL
LIN {X 0,Y 263.081,Z 458.878,A -85,B 0,C 180,E1 -18273.063,E2 -18273.063} C_VEL
LIN {X 0,Y 263.01,Z 460.512,A -85,B 0,C 180,E1 -18274.599,E2 -18274.599} C_VEL
LIN {X 0,Y 262.978,Z 461.764,A -85,B 0,C 180,E1 -18276.137,E2 -18276.137} C_VEL
LIN {X 0,Y 263.019,Z 462.944,A -85,B 0,C 180,E1 -18278.633,E2 -18278.633} C_VEL
LIN {X 0,Y 263.221,Z 463.128,A -85,B 0,C 180,E1 -18280.772,E2 -18280.772} C_VEL
LIN {X 0,Y 263.526,Z 462.809,A -85,B 0,C 180,E1 -18282.319,E2 -18282.319} C_VEL
LIN {X 0,Y 263.922,Z 462.092,A -85,B 0,C 180,E1 -18283.867,E2 -18283.867} C_VEL
LIN {X 0,Y 264.423,Z 460.937,A -85,B 0,C 180,E1 -18285.414,E2 -18285.414} C_VEL
LIN {X 0,Y 265.443,Z 458.593,A -85,B 0,C 180,E1 -18287.605,E2 -18287.605} C_VEL
LIN {X 0,Y 266.759,Z 454.917,A -85,B 0,C 180,E1 -18290.029,E2 -18290.029} C_VEL
LIN {X 0,Y 268.293,Z 450.265,A -85,B 0,C 180,E1 -18292.323,E2 -18292.323} C_VEL
LIN {X 0,Y 270.21,Z 444.318,A -85,B 0,C 180,E1 -18294.592,E2 -18294.592} C_VEL
LIN {X 0,Y 272.354,Z 436.866,A -85,B 0,C 180,E1 -18296.845,E2 -18296.845} C_VEL
LIN {X 0,Y 274.444,Z 429.19,A -85,B 0,C 180,E1 -18298.695,E2 -18298.695} C_VEL
LIN {X 0,Y 276.527,Z 419.747,A -85,B 0,C 180,E1 -18300.551,E2 -18300.551} C_VEL
LIN {X 0,Y 278.695,Z 409.173,A -85,B 0,C 180,E1 -18302.189,E2 -18302.189} C_VEL
LIN {X 0,Y 280.371,Z 398.91,A -85,B 0,C 180,E1 -18303.468,E2 -18303.468} C_VEL
LIN {X 0,Y 281.891,Z 387.533,A -85,B 0,C 180,E1 -18304.576,E2 -18304.576} C_VEL
LIN {X 0,Y 283.001,Z 375.252,A -85,B 0,C 180,E1 -18305.471,E2 -18305.471} C_VEL
LIN {X 0,Y 283.628,Z 363.52,A -85,B 0,C 180,E1 -18306.076,E2 -18306.076} C_VEL
LIN {X 0,Y 284.061,Z 343.9,A -85,B 0,C 180,E1 -18306.676,E2 -18306.676} C_VEL
LIN {X 0,Y 285.046,Z 312.416,A -85,B 0,C 180,E1 -18307.479,E2 -18307.479} C_VEL
LIN {X 0,Y 276.714,Z 296.098,A -85,B 0,C 180,E1 -18309.139,E2 -18309.139} C_VEL
LIN {X 0,Y 267.5,Z 280.643,A -85,B 0,C 180,E1 -18311.061,E2 -18311.061} C_VEL
LIN {X 0,Y 264.904,Z 276.627,A -85,B 0,C 180,E1 -18311.624,E2 -18311.624} C_VEL
LIN {X 0,Y 263.315,Z 273.771,A -85,B 0,C 180,E1 -18312.022,E2 -18312.022} C_VEL
LIN {X 0,Y 263.115,Z 272.782,A -85,B 0,C 180,E1 -18312.38,E2 -18312.38} C_VEL
LIN {X 0,Y 263.078,Z 272.692,A -85,B 0,C 180,E1 -18316.161,E2 -18316.161} C_VEL
LIN {X 0,Y 263.113,Z 272.692,A -85,B 0,C 180,E1 -18320.77,E2 -18320.77} C_VEL
LIN {X 0,Y 263.155,Z 272.683,A -85,B 0,C 180,E1 -18324.016,E2 -18324.016} C_VEL
LIN {X 0,Y 263.125,Z 272.684,A -85,B 0,C 180,E1 -18327.71,E2 -18327.71} C_VEL
LIN {X 0,Y 263.141,Z 272.687,A -85,B 0,C 180,E1 -18331.807,E2 -18331.807} C_VEL
LIN {X 0,Y 263.188,Z 272.687,A -85,B 0,C 180,E1 -18335.217,E2 -18335.217} C_VEL
LIN {X 0,Y 263.248,Z 272.649,A -85,B 0,C 180,E1 -18339.692,E2 -18339.692} C_VEL
LIN {X 0,Y 263.343,Z 272.671,A -85,B 0,C 180,E1 -18344.521,E2 -18344.521} C_VEL
LIN {X 0,Y 263.35,Z 272.674,A -85,B 0,C 180,E1 -18349.233,E2 -18349.233} C_VEL
LIN {X 0,Y 263.522,Z 272.654,A -85,B 0,C 180,E1 -18352.337,E2 -18352.337} C_VEL
LIN {X 0,Y 263.337,Z 272.669,A -85,B 0,C 180,E1 -18355.299,E2 -18355.299} C_VEL
LIN {X 0,Y 262.706,Z 272.751,A -85,B 0,C 180,E1 -18356.578,E2 -18356.578} C_VEL
LIN {X 0,Y 260.088,Z 273.087,A -85,B 0,C 180,E1 -18358.672,E2 -18358.672} C_VEL
LIN {X 0,Y 256.992,Z 273.459,A -85,B 0,C 180,E1 -18361.242,E2 -18361.242} C_VEL
LIN {X 0,Y 256.584,Z 273.506,A -85,B 0,C 180,E1 -18362.128,E2 -18362.128} C_VEL
LIN {X 0,Y 256.45,Z 273.53,A -85,B 0,C 180,E1 -18366.293,E2 -18366.293} C_VEL
LIN {X 0,Y 256.4,Z 273.542,A -85,B 0,C 180,E1 -18369.466,E2 -18369.466} C_VEL
LIN {X 0,Y 256.232,Z 273.557,A -85,B 0,C 180,E1 -18374.291,E2 -18374.291} C_VEL
LIN {X 0,Y 256.177,Z 273.565,A -85,B 0,C 180,E1 -18377.564,E2 -18377.564} C_VEL
LIN {X 0,Y 256.138,Z 273.575,A -85,B 0,C 180,E1 -18381.109,E2 -18381.109} C_VEL
LIN {X 0,Y 256.127,Z 273.575,A -85,B 0,C 180,E1 -18385.11,E2 -18385.11} C_VEL
LIN {X 0,Y 256.038,Z 273.58,A -85,B 0,C 180,E1 -18389.609,E2 -18389.609} C_VEL
LIN {X 0,Y 256.063,Z 273.565,A -85,B 0,C 180,E1 -18393.293,E2 -18393.293} C_VEL
LIN {X 0,Y 256.114,Z 273.577,A -85,B 0,C 180,E1 -18397.271,E2 -18397.271} C_VEL
LIN {X 0,Y 256.017,Z 273.599,A -85,B 0,C 180,E1 -18401.211,E2 -18401.211} C_VEL
LIN {X 0,Y 256.051,Z 273.776,A -85,B 0,C 180,E1 -18404.438,E2 -18404.438} C_VEL
LIN {X 0,Y 259.123,Z 283.731,A -85,B 0,C 180,E1 -18408.233,E2 -18408.233} C_VEL
LIN {X 0,Y 261.702,Z 293.037,A -85,B 0,C 180,E1 -18411.46,E2 -18411.46} C_VEL
LIN {X 0,Y 263.989,Z 302.573,A -85,B 0,C 180,E1 -18414.529,E2 -18414.529} C_VEL
LIN {X 0,Y 264.907,Z 306.766,A -85,B 0,C 180,E1 -18415.735,E2 -18415.735} C_VEL
LIN {X 0,Y 268.342,Z 315.361,A -85,B 0,C 180,E1 -18416.602,E2 -18416.602} C_VEL
LIN {X 0,Y 272.894,Z 344.092,A -85,B 0,C 180,E1 -18418.197,E2 -18418.197} C_VEL
LIN {X 0,Y 275.936,Z 368.983,A -85,B 0,C 180,E1 -18419.392,E2 -18419.392} C_VEL
LIN {X 0,Y 276.848,Z 379.941,A -85,B 0,C 180,E1 -18419.848,E2 -18419.848} C_VEL
LIN {X 0,Y 275.228,Z 419.588,A -85,B 0,C 180,E1 -18420.889,E2 -18420.889} C_VEL
LIN {X 0,Y 273.989,Z 433.063,A -85,B 0,C 180,E1 -18421.514,E2 -18421.514} C_VEL
LIN {X 0,Y 272.192,Z 446.043,A -85,B 0,C 180,E1 -18422.41,E2 -18422.41} C_VEL
LIN {X 0,Y 269.867,Z 457.859,A -85,B 0,C 180,E1 -18423.514,E2 -18423.514} C_VEL
LIN {X 0,Y 267.265,Z 469.267,A -85,B 0,C 180,E1 -18424.911,E2 -18424.911} C_VEL
LIN {X 0,Y 264.629,Z 479.595,A -85,B 0,C 180,E1 -18426.524,E2 -18426.524} C_VEL
LIN {X 0,Y 262.088,Z 488.916,A -85,B 0,C 180,E1 -18428.364,E2 -18428.364} C_VEL
LIN {X 0,Y 259.533,Z 498.027,A -85,B 0,C 180,E1 -18430.626,E2 -18430.626} C_VEL
LIN {X 0,Y 257.497,Z 505.52,A -85,B 0,C 180,E1 -18432.971,E2 -18432.971} C_VEL
LIN {X 0,Y 256.355,Z 510.488,A -85,B 0,C 180,E1 -18434.903,E2 -18434.903} C_VEL
LIN {X 0,Y 255.255,Z 515.452,A -85,B 0,C 180,E1 -18437.275,E2 -18437.275} C_VEL
LIN {X 0,Y 254.657,Z 519.327,A -85,B 0,C 180,E1 -18439.666,E2 -18439.666} C_VEL
LIN {X 0,Y 254.571,Z 522.216,A -85,B 0,C 180,E1 -18442.065,E2 -18442.065} C_VEL
LIN {X 0,Y 254.741,Z 523.629,A -85,B 0,C 180,E1 -18443.664,E2 -18443.664} C_VEL
LIN {X 0,Y 254.881,Z 524.629,A -85,B 0,C 180,E1 -18445.254,E2 -18445.254} C_VEL
LIN {X 0,Y 255.169,Z 525.199,A -85,B 0,C 180,E1 -18446.842,E2 -18446.842} C_VEL
LIN {X 0,Y 255.329,Z 525.339,A -85,B 0,C 180,E1 -18448.422,E2 -18448.422} C_VEL
LIN {X 0,Y 255.453,Z 525.071,A -85,B 0,C 180,E1 -18449.999,E2 -18449.999} C_VEL
LIN {X 0,Y 255.387,Z 524.373,A -85,B 0,C 180,E1 -18451.576,E2 -18451.576} C_VEL
LIN {X 0,Y 255.325,Z 523.22,A -85,B 0,C 180,E1 -18453.155,E2 -18453.155} C_VEL
LIN {X 0,Y 254.958,Z 520.633,A -85,B 0,C 180,E1 -18455.536,E2 -18455.536} C_VEL
LIN {X 0,Y 254.753,Z 516.987,A -85,B 0,C 180,E1 -18457.928,E2 -18457.928} C_VEL
LIN {X 0,Y 254.833,Z 512.203,A -85,B 0,C 180,E1 -18460.326,E2 -18460.326} C_VEL
LIN {X 0,Y 255.432,Z 504.998,A -85,B 0,C 180,E1 -18463.119,E2 -18463.119} C_VEL
LIN {X 0,Y 256.391,Z 497.222,A -85,B 0,C 180,E1 -18465.5,E2 -18465.5} C_VEL
LIN {X 0,Y 257.656,Z 489.307,A -85,B 0,C 180,E1 -18467.459,E2 -18467.459} C_VEL
LIN {X 0,Y 259.18,Z 479.638,A -85,B 0,C 180,E1 -18469.4,E2 -18469.4} C_VEL
LIN {X 0,Y 260.926,Z 468.948,A -85,B 0,C 180,E1 -18471.115,E2 -18471.115} C_VEL
LIN {X 0,Y 262.775,Z 457.047,A -85,B 0,C 180,E1 -18472.609,E2 -18472.609} C_VEL
LIN {X 0,Y 264.404,Z 444.283,A -85,B 0,C 180,E1 -18473.808,E2 -18473.808} C_VEL
LIN {X 0,Y 265.583,Z 431.507,A -85,B 0,C 180,E1 -18474.683,E2 -18474.683} C_VEL
LIN {X 0,Y 266.394,Z 418.972,A -85,B 0,C 180,E1 -18475.243,E2 -18475.243} C_VEL
LIN {X 0,Y 267.378,Z 376.167,A -85,B 0,C 180,E1 -18476.396,E2 -18476.396} C_VEL
LIN {X 0,Y 263.626,Z 333.804,A -85,B 0,C 180,E1 -18477.952,E2 -18477.952} C_VEL
LIN {X 0,Y 260.874,Z 309.716,A -85,B 0,C 180,E1 -18478.955,E2 -18478.955} C_VEL
LIN {X 0,Y 260.971,Z 308.065,A -85,B 0,C 180,E1 -18479.215,E2 -18479.215} C_VEL
LIN {X 0,Y 261.931,Z 300.465,A -85,B 0,C 180,E1 -18481.096,E2 -18481.096} C_VEL
LIN {X 0,Y 259.789,Z 289.216,A -85,B 0,C 180,E1 -18484.229,E2 -18484.229} C_VEL
LIN {X 0,Y 257.174,Z 277.817,A -85,B 0,C 180,E1 -18487.58,E2 -18487.58} C_VEL
LIN {X 0,Y 256.085,Z 273.649,A -85,B 0,C 180,E1 -18488.956,E2 -18488.956} C_VEL
LIN {X 0,Y 256.022,Z 273.578,A -85,B 0,C 180,E1 -18493.333,E2 -18493.333} C_VEL
LIN {X 0,Y 256.027,Z 273.59,A -85,B 0,C 180,E1 -18497.827,E2 -18497.827} C_VEL
LIN {X 0,Y 256.06,Z 273.582,A -85,B 0,C 180,E1 -18500.856,E2 -18500.856} C_VEL
LIN {X 0,Y 256.118,Z 273.576,A -85,B 0,C 180,E1 -18502.866,E2 -18502.866} C_VEL
LIN {X 0,Y 256.058,Z 273.578,A -85,B 0,C 180,E1 -18506.706,E2 -18506.706} C_VEL
LIN {X 0,Y 256.035,Z 273.589,A -85,B 0,C 180,E1 -18510.391,E2 -18510.391} C_VEL
LIN {X 0,Y 256.124,Z 273.57,A -85,B 0,C 180,E1 -18514.888,E2 -18514.888} C_VEL
LIN {X 0,Y 256.115,Z 273.581,A -85,B 0,C 180,E1 -18519.101,E2 -18519.101} C_VEL
LIN {X 0,Y 256.222,Z 273.563,A -85,B 0,C 180,E1 -18524.08,E2 -18524.08} C_VEL
LIN {X 0,Y 256.281,Z 273.55,A -85,B 0,C 180,E1 -18528.933,E2 -18528.933} C_VEL
LIN {X 0,Y 256.458,Z 273.53,A -85,B 0,C 180,E1 -18532.125,E2 -18532.125} C_VEL
LIN {X 0,Y 256.443,Z 273.535,A -85,B 0,C 180,E1 -18536.858,E2 -18536.858} C_VEL
LIN {X 0,Y 256.686,Z 273.496,A -85,B 0,C 180,E1 -18538.431,E2 -18538.431} C_VEL
LIN {X 0,Y 256.687,Z 273.504,A -85,B 0,C 180,E1 -18541.569,E2 -18541.569} C_VEL
LIN {X 0,Y 256.423,Z 273.533,A -85,B 0,C 180,E1 -18546.686,E2 -18546.686} C_VEL
LIN {X 0,Y 256.391,Z 273.533,A -85,B 0,C 180,E1 -18549.467,E2 -18549.467} C_VEL
LIN {X 0,Y 256.223,Z 273.566,A -85,B 0,C 180,E1 -18554.292,E2 -18554.292} C_VEL
LIN {X 0,Y 256.154,Z 273.559,A -85,B 0,C 180,E1 -18557.566,E2 -18557.566} C_VEL
LIN {X 0,Y 256.112,Z 273.58,A -85,B 0,C 180,E1 -18561.098,E2 -18561.098} C_VEL
LIN {X 0,Y 256.076,Z 273.576,A -85,B 0,C 180,E1 -18565.089,E2 -18565.089} C_VEL
LIN {X 0,Y 256.069,Z 273.587,A -85,B 0,C 180,E1 -18568.57,E2 -18568.57} C_VEL
LIN {X 0,Y 256.064,Z 273.586,A -85,B 0,C 180,E1 -18571.701,E2 -18571.701} C_VEL
LIN {X 0,Y 256.073,Z 273.582,A -85,B 0,C 180,E1 -18575.195,E2 -18575.195} C_VEL
LIN {X 0,Y 256.06,Z 273.585,A -85,B 0,C 180,E1 -18579.145,E2 -18579.145} C_VEL
LIN {X 0,Y 255.999,Z 273.557,A -85,B 0,C 180,E1 -18583.341,E2 -18583.341} C_VEL
LIN {X 0,Y 256.031,Z 273.594,A -85,B 0,C 180,E1 -18587.83,E2 -18587.83} C_VEL
LIN {X 0,Y 256.062,Z 273.577,A -85,B 0,C 180,E1 -18590.858,E2 -18590.858} C_VEL
LIN {X 0,Y 256.077,Z 273.578,A -85,B 0,C 180,E1 -18594.808,E2 -18594.808} C_VEL
LIN {X 0,Y 256.076,Z 273.576,A -85,B 0,C 180,E1 -18598.572,E2 -18598.572} C_VEL
LIN {X 0,Y 256.077,Z 273.588,A -85,B 0,C 180,E1 -18602.19,E2 -18602.19} C_VEL
LIN {X 0,Y 256.086,Z 273.574,A -85,B 0,C 180,E1 -18605.692,E2 -18605.692} C_VEL
LIN {X 0,Y 256.162,Z 273.804,A -85,B 0,C 180,E1 -18609.047,E2 -18609.047} C_VEL
LIN {X 0,Y 256.486,Z 274.945,A -85,B 0,C 180,E1 -18609.316,E2 -18609.316} C_VEL
LIN {X 0,Y 264.958,Z 293.21,A -85,B 0,C 180,E1 -18610.773,E2 -18610.773} C_VEL
LIN {X 0,Y 269.288,Z 303.945,A -85,B 0,C 180,E1 -18611.506,E2 -18611.506} C_VEL
LIN {X 0,Y 267.97,Z 357.62,A -85,B 0,C 180,E1 -18612.93,E2 -18612.93} C_VEL
LIN {X 0,Y 267.591,Z 369.745,A -85,B 0,C 180,E1 -18613.454,E2 -18613.454} C_VEL
LIN {X 0,Y 267.072,Z 381.772,A -85,B 0,C 180,E1 -18614.255,E2 -18614.255} C_VEL
LIN {X 0,Y 266.068,Z 393.162,A -85,B 0,C 180,E1 -18615.273,E2 -18615.273} C_VEL
LIN {X 0,Y 264.805,Z 404.328,A -85,B 0,C 180,E1 -18616.573,E2 -18616.573} C_VEL
LIN {X 0,Y 263.317,Z 415.67,A -85,B 0,C 180,E1 -18618.258,E2 -18618.258} C_VEL
LIN {X 0,Y 262.084,Z 424.792,A -85,B 0,C 180,E1 -18619.963,E2 -18619.963} C_VEL
LIN {X 0,Y 260.707,Z 433.146,A -85,B 0,C 180,E1 -18621.865,E2 -18621.865} C_VEL
LIN {X 0,Y 259.215,Z 441.304,A -85,B 0,C 180,E1 -18624.165,E2 -18624.165} C_VEL
LIN {X 0,Y 258.242,Z 446.88,A -85,B 0,C 180,E1 -18626.1,E2 -18626.1} C_VEL
LIN {X 0,Y 257.322,Z 452.324,A -85,B 0,C 180,E1 -18628.436,E2 -18628.436} C_VEL
LIN {X 0,Y 256.58,Z 456.618,A -85,B 0,C 180,E1 -18630.785,E2 -18630.785} C_VEL
LIN {X 0,Y 256.022,Z 459.876,A -85,B 0,C 180,E1 -18633.148,E2 -18633.148} C_VEL
LIN {X 0,Y 255.967,Z 461.482,A -85,B 0,C 180,E1 -18634.725,E2 -18634.725} C_VEL
LIN {X 0,Y 255.933,Z 462.709,A -85,B 0,C 180,E1 -18636.307,E2 -18636.307} C_VEL
LIN {X 0,Y 255.978,Z 463.793,A -85,B 0,C 180,E1 -18638.732,E2 -18638.732} C_VEL
LIN {X 0,Y 256.237,Z 463.969,A -85,B 0,C 180,E1 -18641.07,E2 -18641.07} C_VEL
LIN {X 0,Y 256.566,Z 463.625,A -85,B 0,C 180,E1 -18642.659,E2 -18642.659} C_VEL
LIN {X 0,Y 257,Z 462.854,A -85,B 0,C 180,E1 -18644.248,E2 -18644.248} C_VEL
LIN {X 0,Y 257.552,Z 461.672,A -85,B 0,C 180,E1 -18645.836,E2 -18645.836} C_VEL
LIN {X 0,Y 258.558,Z 459.459,A -85,B 0,C 180,E1 -18647.943,E2 -18647.943} C_VEL
LIN {X 0,Y 260.047,Z 455.537,A -85,B 0,C 180,E1 -18650.569,E2 -18650.569} C_VEL
LIN {X 0,Y 261.681,Z 450.821,A -85,B 0,C 180,E1 -18652.919,E2 -18652.919} C_VEL
LIN {X 0,Y 263.708,Z 444.805,A -85,B 0,C 180,E1 -18655.24,E2 -18655.24} C_VEL
LIN {X 0,Y 265.968,Z 437.269,A -85,B 0,C 180,E1 -18657.544,E2 -18657.544} C_VEL
LIN {X 0,Y 268.17,Z 429.474,A -85,B 0,C 180,E1 -18659.432,E2 -18659.432} C_VEL
LIN {X 0,Y 270.374,Z 419.89,A -85,B 0,C 180,E1 -18661.324,E2 -18661.324} C_VEL
LIN {X 0,Y 272.621,Z 409.167,A -85,B 0,C 180,E1 -18662.996,E2 -18662.996} C_VEL
LIN {X 0,Y 274.397,Z 398.693,A -85,B 0,C 180,E1 -18664.296,E2 -18664.296} C_VEL
LIN {X 0,Y 276.076,Z 386.126,A -85,B 0,C 180,E1 -18665.486,E2 -18665.486} C_VEL
LIN {X 0,Y 277.065,Z 374.394,A -85,B 0,C 180,E1 -18666.325,E2 -18666.325} C_VEL
LIN {X 0,Y 277.768,Z 361.379,A -85,B 0,C 180,E1 -18666.954,E2 -18666.954} C_VEL
LIN {X 0,Y 278.752,Z 324.433,A -85,B 0,C 180,E1 -18667.974,E2 -18667.974} C_VEL
LIN {X 0,Y 279.047,Z 314.595,A -85,B 0,C 180,E1 -18668.233,E2 -18668.233} C_VEL
LIN {X 0,Y 270.923,Z 298.788,A -85,B 0,C 180,E1 -18669.925,E2 -18669.925} C_VEL
LIN {X 0,Y 262.708,Z 285.037,A -85,B 0,C 180,E1 -18671.71,E2 -18671.71} C_VEL
LIN {X 0,Y 258.613,Z 278.353,A -85,B 0,C 180,E1 -18672.654,E2 -18672.654} C_VEL
LIN {X 0,Y 256.509,Z 275.354,A -85,B 0,C 180,E1 -18673.149,E2 -18673.149} C_VEL
LIN {X 0,Y 256.13,Z 274.045,A -85,B 0,C 180,E1 -18673.387,E2 -18673.387} C_VEL
LIN {X 0,Y 256.055,Z 273.596,A -85,B 0,C 180,E1 -18673.874,E2 -18673.874} C_VEL
LIN {X 0,Y 256.033,Z 273.571,A -85,B 0,C 180,E1 -18677.828,E2 -18677.828} C_VEL
LIN {X 0,Y 256.065,Z 273.568,A -85,B 0,C 180,E1 -18680.856,E2 -18680.856} C_VEL
LIN {X 0,Y 256.078,Z 273.578,A -85,B 0,C 180,E1 -18684.806,E2 -18684.806} C_VEL
LIN {X 0,Y 256.076,Z 273.548,A -85,B 0,C 180,E1 -18688.57,E2 -18688.57} C_VEL
LIN {X 0,Y 256.085,Z 273.573,A -85,B 0,C 180,E1 -18692.189,E2 -18692.189} C_VEL
LIN {X 0,Y 256.131,Z 273.554,A -85,B 0,C 180,E1 -18695.695,E2 -18695.695} C_VEL
LIN {X 0,Y 256.149,Z 273.525,A -85,B 0,C 180,E1 -18699.103,E2 -18699.103} C_VEL
LIN {X 0,Y 256.293,Z 273.553,A -85,B 0,C 180,E1 -18704.084,E2 -18704.084} C_VEL
LIN {X 0,Y 256.293,Z 273.557,A -85,B 0,C 180,E1 -18708.933,E2 -18708.933} C_VEL
LIN {X 0,Y 256.464,Z 273.529,A -85,B 0,C 180,E1 -18712.124,E2 -18712.124} C_VEL
